           // --------------------------------------------------------
           // STEP 0
           // Калібровка неактивна
           // --------------------------------------------------------
       UINT#0:

           #qx_BlockForward := FALSE;
           #qx_BlockBackward := FALSE;

           IF #StartEdge THEN

               #stat_Calibrated := FALSE;
               #stat_MotionStarted := FALSE;
               #stat_CompletedSteps := DWORD#0;

               // Очищення даних нової процедури калібровки.
               #stat_RawAtReference := DINT#0;
               #stat_RawAtReferenceValid := FALSE;
               #stat_TravelAfterReference_mm := 0.0;

               // Калібровку можна почати тільки після
               // калібровки підйому та в допустимій зоні.
               IF #HoistPositionOK THEN

                   // Нормальний старт перед репером.
                   IF #ix_Reference3K1 THEN
                       #stat_Step := UINT#10;

                       // Якщо механізм знаходиться на / за 3K1,
                       // спочатку необхідно відійти назад.
                   ELSE
                       #stat_Step := UINT#5;
                   END_IF;

               ELSE

                   #stat_Step := UINT#910;

               END_IF;

           END_IF;


           // --------------------------------------------------------
           // STEP 5
           // Попередній відхід назад від 3K1
           // --------------------------------------------------------
       UINT#5:

           #qx_Active := TRUE;

           #qx_BlockForward := TRUE;
           #qx_BlockBackward := FALSE;

           IF #ix_BtnBackward THEN
               #stat_MotionStarted := TRUE;
           END_IF;

           // Після звільнення 3K1 та відпускання кнопки
           // починаємо стандартну процедуру.
           IF #ix_Reference3K1
               AND NOT #ix_BtnBackward
           THEN

               #stat_Step := UINT#10;

           END_IF;


           // --------------------------------------------------------
           // STEP 10
           // Перевірка початкових умов
           // --------------------------------------------------------
       UINT#10:

           #qx_Active := TRUE;

           IF NOT #ix_BtnForward
               AND NOT #ix_BtnBackward
           THEN

               #stat_CompletedSteps.%X0 := TRUE;
               #stat_Step := UINT#20;

           END_IF;


           // --------------------------------------------------------
           // STEP 20
           // Очікування першої команди "Вперед"
           // --------------------------------------------------------
       UINT#20:

           #qx_Active := TRUE;

           #qx_BlockForward := FALSE;
           #qx_BlockBackward := TRUE;

           IF #ix_BtnForward THEN

               #stat_MotionStarted := TRUE;
               #stat_CompletedSteps.%X1 := TRUE;

               #stat_Step := UINT#30;

           END_IF;


           // --------------------------------------------------------
           // STEP 30
           // Перший рух вперед до 3K1
           // --------------------------------------------------------
       UINT#30:

           #qx_Active := TRUE;

           #qx_BlockForward := FALSE;
           #qx_BlockBackward := TRUE;

           IF #ReferenceFalling THEN

               #stat_CompletedSteps.%X2 := TRUE;
               #stat_Step := UINT#40;

           END_IF;


           // --------------------------------------------------------
           // STEP 40
           // Перше проходження 3K1
           // Очікування відпускання кнопки "Вперед"
           // --------------------------------------------------------
       UINT#40:

           #qx_Active := TRUE;

           #qx_BlockForward := TRUE;
           #qx_BlockBackward := TRUE;

           IF NOT #ix_BtnForward THEN

               #stat_CompletedSteps.%X3 := TRUE;
               #stat_Step := UINT#50;

           END_IF;


           // --------------------------------------------------------
           // STEP 50
           // Відхід назад від репера
           // --------------------------------------------------------
       UINT#50:

           #qx_Active := TRUE;

           #qx_BlockForward := TRUE;
           #qx_BlockBackward := FALSE;

           IF #ix_BtnBackward THEN
               #stat_MotionStarted := TRUE;
           END_IF;

           IF #ix_Reference3K1
               AND NOT #ix_BtnBackward
           THEN

               #stat_CompletedSteps.%X4 := TRUE;
               #stat_Step := UINT#60;

           END_IF;


           // --------------------------------------------------------
           // STEP 60
           // Репер звільнений
           // --------------------------------------------------------
       UINT#60:

           #qx_Active := TRUE;

           #qx_BlockForward := TRUE;
           #qx_BlockBackward := TRUE;

           #stat_CompletedSteps.%X5 := TRUE;
           #stat_Step := UINT#70;


           // --------------------------------------------------------
           // STEP 70
           // Очікування повторної команди "Вперед"
           // --------------------------------------------------------
       UINT#70:

           #qx_Active := TRUE;

           #qx_BlockForward := FALSE;
           #qx_BlockBackward := TRUE;

           IF #ix_BtnForward THEN

               #stat_CompletedSteps.%X6 := TRUE;
               #stat_Step := UINT#80;

           END_IF;


           // --------------------------------------------------------
           // STEP 80
           // Повторний точний підхід до 3K1
           // --------------------------------------------------------
       UINT#80:

           #qx_Active := TRUE;

           #qx_BlockForward := FALSE;
           #qx_BlockBackward := TRUE;

           IF #ReferenceFalling THEN

               // У момент спадного фронту 3K1 запам'ятовуємо
               // фактичне raw-положення енкодера.
               IF #ix_PositionScaleValid THEN

                   #stat_RawAtReference :=
                   #id_ActualPositionRaw;

                   #stat_RawAtReferenceValid :=
                   TRUE;

                   #stat_CompletedSteps.%X7 :=
                   TRUE;

                   #stat_Step :=
                   UINT#90;

               ELSE

                   // Масштабування положення невалідне.
                   #stat_RawAtReferenceValid :=
                   FALSE;

                   #stat_Step :=
                   UINT#910;

               END_IF;

           END_IF;



           // --------------------------------------------------------
           // STEP 90
           // Quick Stop
           // --------------------------------------------------------
       UINT#90:

           #qx_Active := TRUE;

           #qx_BlockForward := TRUE;
           #qx_BlockBackward := TRUE;
           #qx_QuickStop := TRUE;

           #stat_CompletedSteps.%X8 := TRUE;

           #stat_Step := UINT#100;


           // --------------------------------------------------------
           // STEP 100
           // Очікування повної зупинки ПЧ
           // --------------------------------------------------------
       UINT#100:

           #qx_Active := TRUE;

           #qx_BlockForward := TRUE;
           #qx_BlockBackward := TRUE;

           // Quick Stop утримується до підтвердженої зупинки.
           #qx_QuickStop := TRUE;

           IF #qx_DriveStandstill
               AND NOT #ix_BtnForward
               AND NOT #ix_BtnBackward
           THEN

               // Для розрахунку повинна бути зафіксована
               // точка 3K1 і валідне масштабування.
               IF #stat_RawAtReferenceValid
                   AND #ix_PositionScaleValid
               THEN

                   // Розрахунок шляху, пройденого від моменту
                   // спрацювання 3K1 до повної зупинки.
                   #stat_TravelAfterReference_mm :=
                   (
                   DINT_TO_LREAL(#id_ActualPositionRaw)
                   - DINT_TO_LREAL(#stat_RawAtReference)
                   )
                   * #il_Scale_mm_per_count;

                   #stat_CompletedSteps.%X9 :=
                   TRUE;

                   #stat_Step :=
                   UINT#110;

               ELSE

                   // Немає валідної реперної точки
                   // або масштабування положення.
                   #stat_Step :=
                   UINT#910;

               END_IF;

           END_IF;



           // --------------------------------------------------------
           // STEP 110
           // Запуск preset
           // --------------------------------------------------------
       UINT#110:

           #qx_Active := TRUE;

           #qx_BlockForward := TRUE;
           #qx_BlockBackward := TRUE;

           #qx_PresetServiceEnable := TRUE;

           #qx_PresetPermit :=
           #qx_DriveStandstill
           AND NOT #ix_BtnForward
           AND NOT #ix_BtnBackward
           AND #ix_EncoderReady
           AND NOT #ix_EncoderFault
           AND NOT #ix_DriveFault;

           IF #qx_PresetPermit THEN

               #qx_PresetStart := TRUE;

               #stat_CompletedSteps.%X10 := TRUE;
               #stat_Step := UINT#120;

           END_IF;


           // --------------------------------------------------------
           // STEP 120
           // Очікування завершення preset
           // --------------------------------------------------------
       UINT#120:

           #qx_Active := TRUE;

           #qx_BlockForward := TRUE;
           #qx_BlockBackward := TRUE;

           #qx_PresetServiceEnable := TRUE;

           #qx_PresetPermit :=
           #qx_DriveStandstill
           AND NOT #ix_BtnForward
           AND NOT #ix_BtnBackward
           AND NOT #ix_EncoderFault
           AND NOT #ix_DriveFault;

           IF #ix_PresetDone THEN

               #stat_CompletedSteps.%X11 := TRUE;
               #stat_Step := UINT#130;

           ELSIF #ix_PresetError THEN

               #stat_Step := UINT#910;

           END_IF;


           // --------------------------------------------------------
           // STEP 130
           // Калібровка успішно завершена
           // --------------------------------------------------------
       UINT#130:

           #qx_BlockForward := FALSE;
           #qx_BlockBackward := FALSE;

           #stat_Calibrated := TRUE;
           #stat_CompletedSteps.%X12 := TRUE;


           // --------------------------------------------------------
           // STEP 900
           // Ручне переривання
           // --------------------------------------------------------
       UINT#900:

           #qx_Aborted := TRUE;

           #qx_BlockForward := TRUE;
           #qx_BlockBackward := TRUE;

           #qx_QuickStop := TRUE;


           // --------------------------------------------------------
           // STEP 910
           // Помилка процедури
           // --------------------------------------------------------
       UINT#910:

           #qx_Fault := TRUE;

           #qx_BlockForward := TRUE;
           #qx_BlockBackward := TRUE;

           #qx_QuickStop := TRUE;


       ELSE

           #stat_Step := UINT#910;

   END_CASE;


   // ============================================================
   // 11. Основні статуси
   // ============================================================

   #qu_CurrentStep :=
   #stat_Step;

   #qd_CompletedSteps :=
   #stat_CompletedSteps;

   #qx_Calibrated :=
   #stat_Calibrated
   OR #ix_ForceCalibrated;

   // Шлях від повторного проходження 3K1
   // до підтвердженої повної зупинки.
   #ql_TravelAfterReference_mm :=
   #stat_TravelAfterReference_mm;

   // ============================================================
   // 12. Активний таймер для HMI
   // ============================================================

   #qt_ActiveTimerElapsed := T#0ms;
   #qt_ActiveTimerPreset := T#0ms;
   #qt_ActiveTimerRemaining := T#0ms;

   // Timeout A
   IF (#stat_Step = UINT#5)
       OR (#stat_Step = UINT#20)
       OR (#stat_Step = UINT#50)
       OR (#stat_Step = UINT#70)
   THEN

       #qt_ActiveTimerElapsed :=
       #tmr_TimeoutA.ET;

       #qt_ActiveTimerPreset :=
       #it_TimeoutA;

       IF #tmr_TimeoutA.ET < #it_TimeoutA THEN

           #qt_ActiveTimerRemaining :=
           #it_TimeoutA - #tmr_TimeoutA.ET;

       END_IF;


       // Timeout B
   ELSIF 
       (#stat_Step = UINT#30)
       OR (#stat_Step = UINT#80)
   THEN

       #qt_ActiveTimerElapsed :=
       #tmr_TimeoutB.ET;

       #qt_ActiveTimerPreset :=
       #it_TimeoutB;

       IF #tmr_TimeoutB.ET < #it_TimeoutB THEN

           #qt_ActiveTimerRemaining :=
           #it_TimeoutB - #tmr_TimeoutB.ET;

       END_IF;


       // Standstill
   ELSIF #stat_Step = UINT#100 THEN

       #qt_ActiveTimerElapsed :=
       #tmr_Standstill.ET;

       #qt_ActiveTimerPreset :=
       #it_StandstillConfirm;

       IF #tmr_Standstill.ET < #it_StandstillConfirm THEN

           #qt_ActiveTimerRemaining :=
           #it_StandstillConfirm - #tmr_Standstill.ET;

       END_IF;

   END_IF;


   // ============================================================
   // 13. Діагностичне слово
   // ============================================================

   #qw_Status := W#16#0000;

   IF #qx_Active THEN
       #qw_Status := #qw_Status OR W#16#0001;
   END_IF;

   IF #qx_Calibrated THEN
       #qw_Status := #qw_Status OR W#16#0002;
   END_IF;

   IF #qx_Aborted THEN
       #qw_Status := #qw_Status OR W#16#0004;
   END_IF;

   IF #qx_Fault THEN
       #qw_Status := #qw_Status OR W#16#0008;
   END_IF;

   IF #qx_DriveStandstill THEN
       #qw_Status := #qw_Status OR W#16#0010;
   END_IF;

   IF #ix_PresetBusy THEN
       #qw_Status := #qw_Status OR W#16#0020;
   END_IF;

   IF #ix_PresetError THEN
       #qw_Status := #qw_Status OR W#16#0040;
   END_IF;

   IF #tmr_TimeoutA.Q THEN
       #qw_Status := #qw_Status OR W#16#0100;
   END_IF;

   IF #tmr_TimeoutB.Q THEN
       #qw_Status := #qw_Status OR W#16#0200;
   END_IF;

   IF #ix_DriveFault THEN
       #qw_Status := #qw_Status OR W#16#0400;
   END_IF;

   IF #ix_EncoderFault THEN
       #qw_Status := #qw_Status OR W#16#0800;
   END_IF;

   IF NOT #ix_EncoderReady THEN
       #qw_Status := #qw_Status OR W#16#1000;
   END_IF;


   // ============================================================
   // 14. Запам'ятовування станів
   // ============================================================

   #stat_StartOld :=
   #ix_Start;

   #stat_ResetOld :=
   #ix_Reset;

   #stat_AbortOld :=
   #ix_Abort;

   #stat_ReferenceOld :=
   #ix_Reference3K1;
END_FUNCTION_BLOCK

FUNCTION_BLOCK "FB_TrolleyCalibrationDiag"   // FB712, SCL
{ S7_Optimized_Access := 'TRUE' }
VERSION : 0.1
   VAR_INPUT
      ix_Reset : Bool := FALSE;   // Скидання зафіксованих діагностичних помилок
      ix_EncoderReady : Bool := FALSE;   // Енкодер 3BR готовий
      ix_EncoderFault : Bool := FALSE;   // Помилка енкодера
      ix_CommunicationFault : Bool := FALSE;   // Помилка зв'язку з енкодером
      il_Position_mm : LReal := 0.0;   // Поточна координата візка, мм
      ix_MoveCommand : Bool := FALSE;   // Дійсна команда руху візка
      ix_DriveFault : Bool := FALSE;   // Аварія привода
      ir_DriveVelocity_rpm : Real := 0.0;   // Фактична швидкість привода
      ix_CalibrationActive : Bool := FALSE;   // Процедура калібровки візка активна
      ix_Calibrated : Bool := FALSE;   // Візок відкалібрований
      ix_ManualDriveActive : Bool := FALSE;   // Ручний привод активний; поки FALSE
      il_NoMoveThreshold_mm : LReal := 5.0;   // Допустима зміна положення без команди
      il_MoveMinDelta_mm : LReal := 1.0;   // Мінімальна зміна при русі
      it_MoveUpdateTimeout : Time := T#1s;   // Максимальний час без зміни положення
      ir_StandstillSpeed_rpm : Real := 5.0;   // Поріг повної зупинки
      it_StandstillConfirm : Time := T#500ms;   // Час підтвердження повної зупинки
      il_StartupTolerance_mm : LReal := 5.0;   // Допуск після запуску PLC
   END_VAR
   VAR_OUTPUT
      qx_EncoderControlHealthy : Bool := FALSE;   // Енкодер 3BR і зв'язок справні
      qx_StartupDataConsistent : Bool := TRUE;   // Положення після старту PLC узгоджене
      qx_NoMovementWithoutCommand : Bool := TRUE;   // Не виявлено переміщення без команди
      qx_NoManualMovementDetected : Bool := TRUE;   // Не виявлено нештатного руху без ручного приводу
      qx_EncoderUpdatesDuringMotion : Bool := TRUE;   // Енкодер змінює значення при команді руху
      qx_EncoderReplacementNotDetected : Bool := TRUE;   // Зарезервовано; поки завжди норма
      qx_DiagnosticsHealthy : Bool := FALSE;   // Усі реалізовані контролі в нормі
      qx_DriveStandstill : Bool := FALSE;   // Підтверджена повна зупинка
      ql_PositionDeltaStopped_mm : LReal := 0.0;   // Зміна позиції від точки зупинки
      ql_PositionDeltaMotion_mm : LReal := 0.0;   // Зміна позиції для watchdog руху
   END_VAR
   VAR RETAIN
      stat_SavedPosition_mm : LReal := 0.0;   // Положення, збережене до перезапуску
      stat_SavedPositionValid : Bool := FALSE;   // Ознака валідності збереженого положення
   END_VAR
   VAR
      stat_StartupChecked : Bool := FALSE;   // Перевірка після запуску PLC виконана
      stat_StopReference_mm : LReal := 0.0;   // Базова позиція після зупинки
      stat_StopReferenceValid : Bool := FALSE;   // Базова позиція зупинки валідна
      stat_MoveReference_mm : LReal := 0.0;   // Базова позиція для watchdog руху
      stat_MoveMonitorActive : Bool := FALSE;   // Контроль зміни позиції при русі активний
      stat_WasMoving : Bool := FALSE;   // Ознака, що механізм до цього рухався
      stat_StartupMismatchFault : Bool := FALSE;   // Виявлена невідповідність положення після запуску
      stat_MoveWithoutCommandFault : Bool := FALSE;   // Виявлено зміну положення без команди руху
      stat_NoUpdateDuringMotionFault : Bool := FALSE;   // Не виявлено зміни положення при команді руху
      stat_CalibratedOld : Bool := FALSE;   // Попередній стан сигналу Calibrated
      tmr_Standstill : TON_TIME;   // Таймер підтвердження повної зупинки
      tmr_MoveUpdate : TON_TIME;   // Watchdog оновлення положення при русі
   END_VAR
   VAR_TEMP
      EncoderHealthy : Bool;   // Поточна справність енкодера і зв'язку
      StandstillCondition : Bool;   // Умова низької швидкості
      CalibratedRising : Bool;   // Передній фронт статусу калібровки
      MoveDeltaReached : Bool;   // Досягнута мінімальна зміна положення
      MoveWatchdogEnable : Bool;   // Дозвіл watchdog руху
   END_VAR
BEGIN
       // ============================================================
       // 1. Загальна справність енкодера 3BR
       // ============================================================

       #EncoderHealthy :=
       #ix_EncoderReady
       AND NOT #ix_EncoderFault
       AND NOT #ix_CommunicationFault;

       #qx_EncoderControlHealthy :=
       #EncoderHealthy;


       // ============================================================
       // 2. Визначення повної зупинки
       // ============================================================

       #StandstillCondition :=
       ABS(#ir_DriveVelocity_rpm)
       <= #ir_StandstillSpeed_rpm;

       #tmr_Standstill(
                       IN :=
                       #StandstillCondition
                       AND NOT #ix_MoveCommand,
                       PT := #it_StandstillConfirm
       );

       #qx_DriveStandstill :=
       #tmr_Standstill.Q;


       // ============================================================
       // 3. Фронт отримання статусу "Калібровано"
       // ============================================================

       #CalibratedRising :=
       #ix_Calibrated
       AND NOT #stat_CalibratedOld;


       // ============================================================
       // 4. Reset діагностики
       // ============================================================

       IF #ix_Reset THEN

           #stat_StartupMismatchFault := FALSE;
           #stat_MoveWithoutCommandFault := FALSE;
           #stat_NoUpdateDuringMotionFault := FALSE;

           #stat_StopReferenceValid := FALSE;
           #stat_MoveMonitorActive := FALSE;

       END_IF;


       // ============================================================
       // 5. Перевірка положення після запуску PLC
       //
       // Виконується один раз після появи валідних даних енкодера.
       // Retain-позиція не перезаписується до завершення перевірки.
       // ============================================================

       IF NOT #stat_StartupChecked
           AND #EncoderHealthy
       THEN

           IF #stat_SavedPositionValid THEN

               IF ABS(#il_Position_mm - #stat_SavedPosition_mm)
                   > #il_StartupTolerance_mm
               THEN

                   #stat_StartupMismatchFault := TRUE;

               END_IF;

           ELSE

               // Перший запуск: попереднього значення ще немає.
               #stat_SavedPosition_mm :=
               #il_Position_mm;

               #stat_SavedPositionValid := TRUE;

           END_IF;

           #stat_StartupChecked := TRUE;

           // Початкова база для контролю нерухомості.
           #stat_StopReference_mm :=
           #il_Position_mm;

           #stat_StopReferenceValid := TRUE;

       END_IF;


       // ============================================================
       // 6. Після успішної калібровки
       //
       // Preset штатно змінює координату без фізичного руху.
       // Тому після калібровки формуємо нову базову позицію.
       // ============================================================

       IF #CalibratedRising
           AND #EncoderHealthy
       THEN

           #stat_StopReference_mm :=
           #il_Position_mm;

           #stat_StopReferenceValid := TRUE;

           #stat_SavedPosition_mm :=
           #il_Position_mm;

           #stat_SavedPositionValid := TRUE;

           // Калібровка формує нову достовірну координату.
           #stat_StartupMismatchFault := FALSE;
           #stat_MoveWithoutCommandFault := FALSE;
           #stat_NoUpdateDuringMotionFault := FALSE;

       END_IF;


       // ============================================================
       // 7. Запам'ятовування факту руху
       // ============================================================

       IF #ix_MoveCommand THEN
           #stat_WasMoving := TRUE;
       END_IF;


       // ============================================================
       // 8. Формування нової бази після завершення руху
       //
       // Після підтвердженої повної зупинки зберігаємо положення.
       // ============================================================

       IF #qx_DriveStandstill
           AND #stat_WasMoving
           AND #EncoderHealthy
           AND NOT #ix_CalibrationActive
       THEN

           #stat_StopReference_mm :=
           #il_Position_mm;

           #stat_StopReferenceValid := TRUE;

           #stat_SavedPosition_mm :=
           #il_Position_mm;

           #stat_SavedPositionValid := TRUE;

           #stat_WasMoving := FALSE;

       END_IF;


       // ============================================================
       // 9. Контроль зміни положення без команди руху
       //
       // Контроль виконується тільки:
       // - після підтвердженої повної зупинки;
       // - без команди руху;
       // - без ручного приводу;
       // - поза процедурою калібровки.
       // ============================================================

       #ql_PositionDeltaStopped_mm := 0.0;

       IF #qx_DriveStandstill
           AND NOT #ix_MoveCommand
           AND NOT #ix_ManualDriveActive
           AND NOT #ix_CalibrationActive
           AND #EncoderHealthy
           AND #stat_StopReferenceValid
       THEN

           #ql_PositionDeltaStopped_mm :=
           ABS(#il_Position_mm - #stat_StopReference_mm);

           IF #ql_PositionDeltaStopped_mm
               > #il_NoMoveThreshold_mm
           THEN

               #stat_MoveWithoutCommandFault := TRUE;

           END_IF;

       END_IF;


       // ============================================================
       // 10. Контроль оновлення енкодера під час руху
       //
       // Якщо є дійсна команда руху і немає аварії привода,
       // координата повинна змінюватись не менш ніж на задану
       // величину протягом MoveUpdateTimeout.
       // ============================================================

       IF #ix_MoveCommand
           AND NOT #ix_DriveFault
           AND #EncoderHealthy
       THEN

           IF NOT #stat_MoveMonitorActive THEN

               #stat_MoveReference_mm :=
               #il_Position_mm;

               #stat_MoveMonitorActive := TRUE;

           END_IF;

           #ql_PositionDeltaMotion_mm :=
           ABS(#il_Position_mm - #stat_MoveReference_mm);

           #MoveDeltaReached :=
           #ql_PositionDeltaMotion_mm >= #il_MoveMinDelta_mm;

           IF #MoveDeltaReached THEN

               // Є нормальна зміна координати.
               // Починаємо наступний інтервал контролю.
               #stat_MoveReference_mm :=
               #il_Position_mm;

           END_IF;

       ELSE

           #stat_MoveMonitorActive := FALSE;
           #ql_PositionDeltaMotion_mm := 0.0;
           #MoveDeltaReached := FALSE;

       END_IF;


       // Watchdog працює, поки координата не змінилася
       // на необхідну величину.
       #MoveWatchdogEnable :=
       #stat_MoveMonitorActive
       AND NOT #MoveDeltaReached;

       #tmr_MoveUpdate(
                       IN := #MoveWatchdogEnable,
                       PT := #it_MoveUpdateTimeout
       );

       IF #tmr_MoveUpdate.Q THEN
           #stat_NoUpdateDuringMotionFault := TRUE;
       END_IF;


       // ============================================================
       // 11. Позитивні діагностичні виходи
       // ============================================================

       #qx_StartupDataConsistent :=
       NOT #stat_StartupMismatchFault;

       #qx_NoMovementWithoutCommand :=
       NOT #stat_MoveWithoutCommandFault;

       // Поки окремого сигналу ручного приводу немає.
       // Контроль використовує його як дозвільну умову.
       #qx_NoManualMovementDetected :=
       NOT #stat_MoveWithoutCommandFault;

       #qx_EncoderUpdatesDuringMotion :=
       NOT #stat_NoUpdateDuringMotionFault;


       // ============================================================
       // 12. Контроль фізичної заміни енкодера
       //
       // Поки не реалізований.
       // До появи надійного способу ідентифікації енкодера
       // сигнал примусово встановлений у стан "Норма".
       // ============================================================

       #qx_EncoderReplacementNotDetected := TRUE;


       // ============================================================
       // 13. Загальний результат
       // ============================================================

       #qx_DiagnosticsHealthy :=
       #qx_EncoderControlHealthy
       AND #qx_StartupDataConsistent
       AND #qx_NoMovementWithoutCommand
       AND #qx_NoManualMovementDetected
       AND #qx_EncoderUpdatesDuringMotion;


       // ============================================================
       // 14. Запам'ятовування станів
       // ============================================================

       #stat_CalibratedOld :=
       #ix_Calibrated;
END_FUNCTION_BLOCK

// folder: 70_FireAlarm

FUNCTION_BLOCK "FB_FireAlarm"   // FB70, LAD
TITLE = Пожежна сигналізація
{ S7_Optimized_Access := 'TRUE' }
VERSION : 0.1
   VAR_INPUT
      ix_VFD1_PM_AirIntakeOvertemp : Bool;   // ПЧ1 - Силовий модуль: перегрів повітря на вході
      ix_VFD2_PM_AirIntakeOvertemp : Bool;   // ПЧ2 - Силовий модуль: перегрів повітря на вході
      ix_VFD3_PM_AirIntakeOvertemp : Bool;   // ПЧ3 - Силовий модуль: перегрів повітря на вході
      ix_VFD1_OvertempMonitor : Bool;   // ПЧ1 - Додатковий контроль температури
      ix_VFD2_OvertempMonitor : Bool;   // ПЧ2 - Додатковий контроль температури
      ix_VFD3_OvertempMonitor : Bool;   // ПЧ3 - Додатковий контроль температури
      ix_Ack : Bool;   // Скидання пожежної сигналізації
   END_VAR
   VAR_OUTPUT
      ox_FireAlarmActive : Bool;   // Активна пожежна сигналізація
      ox_SoundFireAlarm : Bool;   // Звукова пожежна сигналізація
   END_VAR
   VAR
      T_FireAlarmDelay : TON_TIME;   // Таймер затримки спрацювання сигналізації
      T_DelaySP : Time := T#30s;   // Уставка часу
      T_SoundAlarm_Active : TON_TIME;   // Таймер видачі звуку
      T_SoundAlarm_Idle : TON_TIME;   // Таймер паузи звуку
      sx_SoundAlarmActive : Bool;   // Активна звукова сигналызація
   END_VAR
   VAR_TEMP
      Condition1 : Bool;   // Умова 1 = ПЧ1+ПЧ2
      Condition2 : Bool;   // Умова 2 = ПЧ1 +ПЧ3
      Condition3 : Bool;   // Умова 3 = ПЧ2 + ПЧ3
   END_VAR
   // T_SoundAlarm_Active.PT := T#3s;
   // T_SoundAlarm_Idle.PT := T#1s;
BEGIN

REGION Network 1: Скидання активної пожежної сигналізації
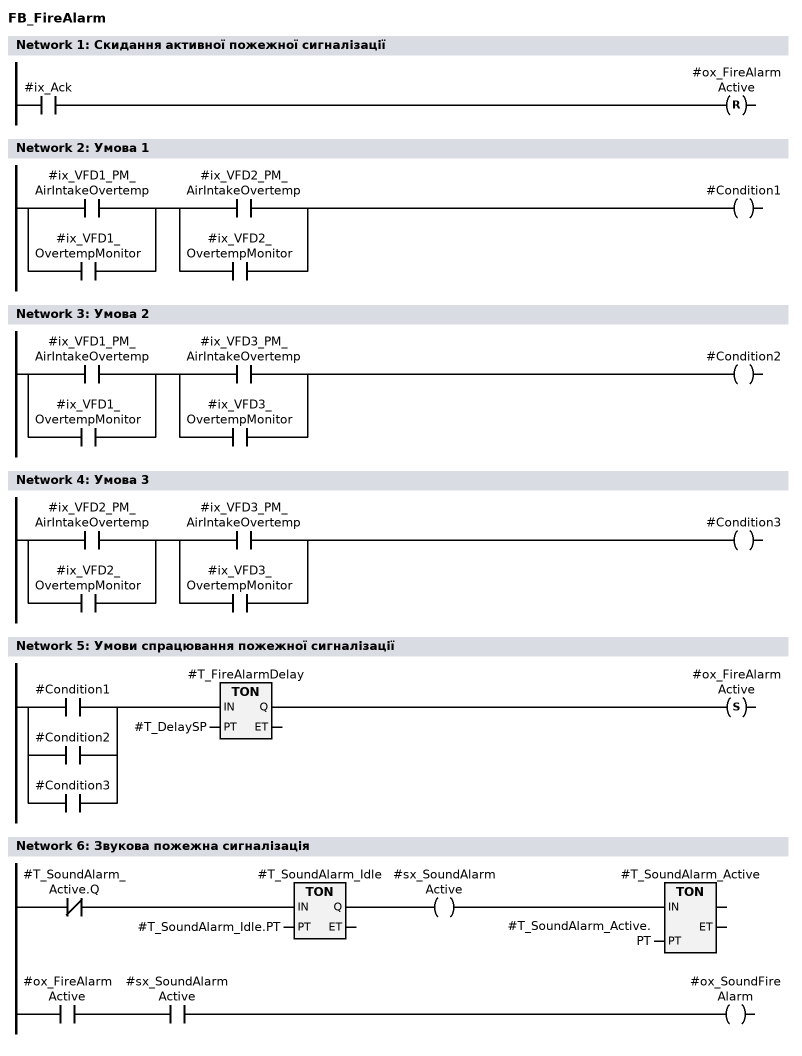
   RUNG wire#powerrail
      Contact( #ix_Ack )
      R_Coil( #ox_FireAlarmActive )
   END_RUNG
   // the same network as SCL:
   IF #ix_Ack THEN #ox_FireAlarmActive := FALSE; END_IF;
END_REGION

REGION Network 2: Умова 1
   RUNG wire#powerrail
      Contact( #ix_VFD1_PM_AirIntakeOvertemp )
      wire#w1
      Contact( #ix_VFD2_PM_AirIntakeOvertemp )
      wire#w2
      Coil( #Condition1 )
   END_RUNG
   RUNG wire#powerrail
      Contact( #ix_VFD1_OvertempMonitor )
   END_RUNG wire#w1
   RUNG wire#w1
      Contact( #ix_VFD2_OvertempMonitor )
   END_RUNG wire#w2
   // the same network as SCL:
   #Condition1 := (#ix_VFD1_PM_AirIntakeOvertemp OR #ix_VFD1_OvertempMonitor) AND (#ix_VFD2_PM_AirIntakeOvertemp OR #ix_VFD2_OvertempMonitor);
END_REGION

REGION Network 3: Умова 2
   RUNG wire#powerrail
      Contact( #ix_VFD1_PM_AirIntakeOvertemp )
      wire#w1
      Contact( #ix_VFD3_PM_AirIntakeOvertemp )
      wire#w2
      Coil( #Condition2 )
   END_RUNG
   RUNG wire#powerrail
      Contact( #ix_VFD1_OvertempMonitor )
   END_RUNG wire#w1
   RUNG wire#w1
      Contact( #ix_VFD3_OvertempMonitor )
   END_RUNG wire#w2
   // the same network as SCL:
   #Condition2 := (#ix_VFD1_PM_AirIntakeOvertemp OR #ix_VFD1_OvertempMonitor) AND (#ix_VFD3_PM_AirIntakeOvertemp OR #ix_VFD3_OvertempMonitor);
END_REGION

REGION Network 4: Умова 3
   RUNG wire#powerrail
      Contact( #ix_VFD2_PM_AirIntakeOvertemp )
      wire#w1
      Contact( #ix_VFD3_PM_AirIntakeOvertemp )
      wire#w2
      Coil( #Condition3 )
   END_RUNG
   RUNG wire#powerrail
      Contact( #ix_VFD2_OvertempMonitor )
   END_RUNG wire#w1
   RUNG wire#w1
      Contact( #ix_VFD3_OvertempMonitor )
   END_RUNG wire#w2
   // the same network as SCL:
   #Condition3 := (#ix_VFD2_PM_AirIntakeOvertemp OR #ix_VFD2_OvertempMonitor) AND (#ix_VFD3_PM_AirIntakeOvertemp OR #ix_VFD3_OvertempMonitor);
END_REGION

REGION Network 5: Умови спрацювання пожежної сигналізації
   #T_FireAlarmDelay(IN := #Condition1 OR #Condition2 OR #Condition3, PT := #T_DelaySP);   // TON
   IF #T_FireAlarmDelay.Q THEN #ox_FireAlarmActive := TRUE; END_IF;
END_REGION

REGION Network 6: Звукова пожежна сигналізація
   #T_SoundAlarm_Idle(IN := NOT #T_SoundAlarm_Active.Q, PT := #T_SoundAlarm_Idle.PT);   // TON
   #sx_SoundAlarmActive := #T_SoundAlarm_Idle.Q;
   #T_SoundAlarm_Active(IN := #T_SoundAlarm_Idle.Q, PT := #T_SoundAlarm_Active.PT);   // TON
   #ox_SoundFireAlarm := #ox_FireAlarmActive AND #sx_SoundAlarmActive;
END_REGION
END_FUNCTION_BLOCK

FUNCTION "FC_FireAlarmCall" : Void   // FC70, LAD
TITLE = Пожежна сигналізація
{ S7_Optimized_Access := 'TRUE' }
VERSION : 0.1
BEGIN

REGION Network 1: Пожежна сигналізація
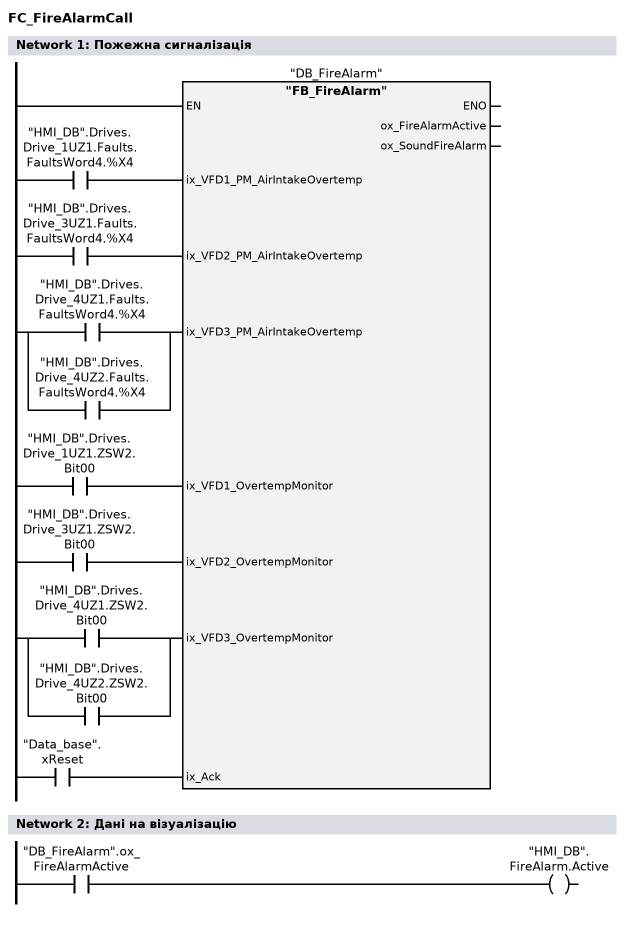
   RUNG wire#powerrail
      "DB_FireAlarm"(ix_VFD1_PM_AirIntakeOvertemp := wire#w1, ix_VFD2_PM_AirIntakeOvertemp := wire#w2, ix_VFD3_PM_AirIntakeOvertemp := wire#w3, ix_VFD1_OvertempMonitor := wire#w4, ix_VFD2_OvertempMonitor := wire#w5, ix_VFD3_OvertempMonitor := wire#w6, ix_Ack := wire#w7, ox_FireAlarmActive =>, ox_SoundFireAlarm =>)
   END_RUNG
   RUNG wire#powerrail
      Contact( "HMI_DB".Drives.Drive_1UZ1.Faults.FaultsWord4.%X4 )
   END_RUNG wire#w1
   RUNG wire#powerrail
      Contact( "HMI_DB".Drives.Drive_3UZ1.Faults.FaultsWord4.%X4 )
   END_RUNG wire#w2
   RUNG wire#powerrail
      Contact( "HMI_DB".Drives.Drive_4UZ1.Faults.FaultsWord4.%X4 )
   END_RUNG wire#w3
   RUNG wire#powerrail
      Contact( "HMI_DB".Drives.Drive_4UZ2.Faults.FaultsWord4.%X4 )
   END_RUNG wire#w3
   RUNG wire#powerrail
      Contact( "HMI_DB".Drives.Drive_1UZ1.ZSW2.Bit00 )
   END_RUNG wire#w4
   RUNG wire#powerrail
      Contact( "HMI_DB".Drives.Drive_3UZ1.ZSW2.Bit00 )
   END_RUNG wire#w5
   RUNG wire#powerrail
      Contact( "HMI_DB".Drives.Drive_4UZ1.ZSW2.Bit00 )
   END_RUNG wire#w6
   RUNG wire#powerrail
      Contact( "HMI_DB".Drives.Drive_4UZ2.ZSW2.Bit00 )
   END_RUNG wire#w6
   RUNG wire#powerrail
      Contact( "Data_base".xReset )
   END_RUNG wire#w7
   // the same network as SCL:
   "DB_FireAlarm"(ix_VFD1_PM_AirIntakeOvertemp := "HMI_DB".Drives.Drive_1UZ1.Faults.FaultsWord4.%X4,   // "FB_FireAlarm"
                  ix_VFD2_PM_AirIntakeOvertemp := "HMI_DB".Drives.Drive_3UZ1.Faults.FaultsWord4.%X4,
                  ix_VFD3_PM_AirIntakeOvertemp := "HMI_DB".Drives.Drive_4UZ1.Faults.FaultsWord4.%X4 OR "HMI_DB".Drives.Drive_4UZ2.Faults.FaultsWord4.%X4,
                  ix_VFD1_OvertempMonitor := "HMI_DB".Drives.Drive_1UZ1.ZSW2.Bit00,
                  ix_VFD2_OvertempMonitor := "HMI_DB".Drives.Drive_3UZ1.ZSW2.Bit00,
                  ix_VFD3_OvertempMonitor := "HMI_DB".Drives.Drive_4UZ1.ZSW2.Bit00 OR "HMI_DB".Drives.Drive_4UZ2.ZSW2.Bit00,
                  ix_Ack := "Data_base".xReset);
END_REGION

REGION Network 2: Дані на візуалізацію
   RUNG wire#powerrail
      Contact( "DB_FireAlarm".ox_FireAlarmActive )
      Coil( "HMI_DB".FireAlarm.Active )
   END_RUNG
   // the same network as SCL:
   "HMI_DB".FireAlarm.Active := "DB_FireAlarm".ox_FireAlarmActive;
END_REGION
END_FUNCTION

// folder: 80_Encoders

FUNCTION_BLOCK "FB_Enc_Tlg89_Com"   // FB80, SCL
{ S7_Optimized_Access := 'TRUE' }
VERSION : 0.1
   VAR_INPUT
      HW_ID_Tlg89 : Hw_Io;   // HW ID підмодуля Standard Telegram 89, PZD3/5. Це має бути HW ID саме телеграмного підмодуля, не головного модуля енкодера.
      Enable : Bool := TRUE;   // Загальний дозвіл роботи блока.
      AckError : Bool := FALSE;   // Квітування помилки енкодера по передньому фронту. Формує STW2_ENC bit 7.
      PresetServiceEnable : Bool := FALSE;   // Дозвіл сервісної функції preset. Для нормальної роботи має бути FALSE.
      PresetPermit : Bool := FALSE;   // Додатковий дозвіл preset від логіки ПЛК. Сюди треба подавати умови: механізм стоїть, сервісний режим активний, немає команд руху.
      PresetStart : Bool := FALSE;   // Команда запуску preset по передньому фронту. Формує STW2_ENC bit 0.
      PresetValueRaw : DInt := DINT#0;   // Значення preset у raw-count. Для 30-bit енкодера допустимий діапазон 0...1073741823.
      SimulationMode : Bool := FALSE;   // Дозвіл режиму симуляції з боку виклику блока.
      SimPzdIn : "UDT_Enc_Tlg89_In";   // Вхідна PZD-структура від симулятора енкодера.
      SimInputValid : Bool := FALSE;   // Ознака, що симуляційні PZD-дані достовірні.
   END_VAR
   VAR_OUTPUT
      AbsolutePositionRaw : DInt := DINT#0;   // Абсолютне положення з G1_XIST2. Використовувати тільки якщо PositionDataValid = TRUE.
      VelocityRaw : DInt := DINT#0;   // Швидкість з NIST_B. Використовувати тільки якщо VelocityDataValid = TRUE.
      PositionDataValid : Bool := FALSE;   // Положення можна використовувати в логіці керування.
      VelocityDataValid : Bool := FALSE;   // Швидкість можна використовувати в логіці керування.
      EncoderReady : Bool := FALSE;   // Фінальна готовність енкодера для логіки крана.
      CommunicationFault : Bool := FALSE;   // Загальна помилка комунікації або недостовірності обміну.
      EncoderFault : Bool := FALSE;   // ZSW2_ENC bit 3. Активна помилка енкодера.
      EncoderAlarm : Bool := FALSE;   // ZSW2_ENC bit 7. Попередження або alarm.
      EncoderErrorCode : DInt := DINT#0;   // Код активної помилки енкодера з G1_XIST2. 0 — активної помилки немає.
      ControlByPlcActive : Bool := FALSE;   // ZSW2_ENC bit 9. Енкодер підтвердив керування / валідність циклічних даних від PLC.
      EncoderLifeValid : Bool := FALSE;   // Encoder sign-of-life валідний.
      PresetBusy : Bool := FALSE;   // TRUE, якщо preset-процедура активна.
      PresetDone : Bool := FALSE;   // Імпульс на один цикл після успішного preset.
      PresetError : Bool := FALSE;   // TRUE, якщо preset-процедура завершилась помилкою.
      PresetStatus : Word := W#16#0000;   // Діагностичний код preset-процедури.
      Status : Word := W#16#0000;   // Загальне діагностичне слово блока.
   END_VAR
   VAR
      SimulationPermit : Bool := FALSE;   // Додатковий дозвіл симуляції. Реальна симуляція активна тільки якщо SimulationMode = TRUE і SimulationPermit = TRUE.
      EnableSignOfLife : Bool := FALSE;   // Дозвіл формування master sign-of-life у STW2_ENC bits 12...15.
      MonitorSignOfLife : Bool := FALSE;   // Дозвіл контролю encoder sign-of-life із ZSW2_ENC bits 12...15.
      MaxUnchangedLifeCycles : UInt := UINT#10;   // Максимальна кількість циклів без зміни encoder sign-of-life.
   END_VAR
   VAR RETAIN
      MaxPositionRaw : DInt := DINT#1073741823;   // Максимальне допустиме raw-значення для 30-bit енкодера.
   END_VAR
   VAR
      PzdIn : "UDT_Enc_Tlg89_In";   // Буфер для DPRD_DAT у реальному режимі.
      PzdOut : "UDT_Enc_Tlg89_Out";   // Буфер для DPWR_DAT у реальному режимі.
      PzdInActual : "UDT_Enc_Tlg89_In";   // Фактично використана вхідна PZD-структура: з енкодера або з симулятора.
      PzdOutActual : "UDT_Enc_Tlg89_Out";   // Фактично сформована вихідна PZD-структура.
      SimPzdOut : "UDT_Enc_Tlg89_Out";   // Вихідна PZD-структура для симулятора. Підключається до входу PzdFromController у симуляційному FB.
      ReadRetVal : Int := INT#0;   // Код повернення DPRD_DAT.
      WriteRetVal : Int := INT#0;   // Код повернення DPWR_DAT.
      ReadError : Bool := FALSE;   // Помилка читання PZD-даних.
      WriteError : Bool := FALSE;   // Помилка запису PZD-даних.
      PresetAck : Bool := FALSE;   // ZSW2_ENC bit 0. Підтвердження виконання preset.
      PositionActualValidBit : Bool := FALSE;   // ZSW2_ENC bit 1. Фактичне положення валідне.
      VelocityActualValidBit : Bool := FALSE;   // ZSW2_ENC bit 2. Фактична швидкість валідна.
      MasterSignOfLife : USInt := USINT#1;   // Поточне значення master sign-of-life, яке PLC передає в STW2_ENC bits 12...15.
      EncoderSignOfLife : USInt := USINT#0;   // Поточне значення encoder sign-of-life із ZSW2_ENC bits 12...15.
      EncoderLifeChanged : Bool := FALSE;   // Encoder sign-of-life змінився в поточному циклі.
      UnchangedLifeCycles : UInt := UINT#0;   // Кількість циклів без зміни encoder sign-of-life.
   END_VAR
   VAR RETAIN
      ActivePresetValueRaw : DInt := DINT#0;   // Значення, яке зараз передається в G1_XIST_PRESET_B1.
   END_VAR
   VAR
      PrevPresetAck : Bool := FALSE;   // Попередній стан ZSW2_ENC bit 0.
      PresetAckRising : Bool := FALSE;   // Передній фронт підтвердження preset від енкодера.
      AckErrorEdge : R_TRIG;   // Формування переднього фронту AckError.
      PresetStartEdge : R_TRIG;   // Формування переднього фронту PresetStart.
      SimulationActive : Bool := FALSE;   // Активний режим симуляції: SimulationMode AND SimulationPermit.
      MasterLifeCounter : USInt := USINT#1;   // Внутрішній лічильник master sign-of-life 1...15.
      LastEncoderLifeCounter : USInt := USINT#0;   // Попереднє значення encoder sign-of-life.
      UnchangedLifeCyclesInt : UInt := UINT#0;   // Внутрішній лічильник циклів без зміни encoder sign-of-life.
      CmdAckError : Bool := FALSE;   // Внутрішній імпульс квітування помилки.
      TempLifeUInt : UInt := UINT#0;   // Тимчасова змінна для виділення encoder sign-of-life.
      TempMasterLifeUInt : UInt := UINT#0;   // Тимчасова змінна для запису master sign-of-life у STW2_ENC.
   END_VAR
   VAR RETAIN
      AckErrorHoldCycles : UInt := UINT#10;   // Кількість циклів утримання STW2_ENC bit 7.
   END_VAR
   VAR
      AckErrorHoldCounter : UInt := UINT#0;   // Поточний лічильник циклів утримання квітування.
   END_VAR
   VAR RETAIN
      PresetTimeoutCycles : UInt := UINT#100;   // Максимальна тривалість очікування preset acknowledgment
   END_VAR
   VAR
      PresetTimeoutCounter : UInt := UINT#0;   // Поточний лічильник очікування
   END_VAR
BEGIN
   //PresetStatus — розшифровка
   //|       Код | Значення                                      |
   //| --------: | --------------------------------------------- |
   //| `16#0000` | Немає помилки.                                |
   //| `16#8201` | `#PresetServiceEnable = FALSE`.                |
   //| `16#8202` | Немає дозволу `PresetPermit`.                 |
   //| `16#8203` | Енкодер не готовий або є помилка комунікації. |
   //| `16#8204` | Preset вже активний.                          |
   //| `16#8205` | `#PresetValueRaw` поза допустимим діапазоном.  |
   //| `16#8206` | Не отримано підтвердження preset протягом заданого часу |


   //Status — діагностичне слово блока
   //| Біт |     Маска | Значення                     |
   //| --: | --------: | ---------------------------- |
   //|   0 | `16#0001` | `#ReadError = TRUE`           |
   //|   1 | `16#0002` | `#WriteError = TRUE`          |
   //|   2 | `16#0004` | `#CommunicationFault = TRUE`  |
   //|   3 | `16#0008` | `#ControlByPlcActive = FALSE` |
   //|   4 | `16#0010` | `#EncoderFault = TRUE`        |
   //|   5 | `16#0020` | `#EncoderAlarm = TRUE`        |
   //|   8 | `16#0100` | `#EncoderLifeValid = FALSE`   |
   //|   9 | `16#0200` | `#PositionDataValid = FALSE`  |
   //|  10 | `16#0400` | `#VelocityDataValid = FALSE`  |
   //|  11 | `16#0800` | `#EncoderReady = FALSE`       |
   //|  12 | `16#1000` | `SimulationActive = TRUE`    |
   //|  13 | `16#2000` | `#PresetBusy = TRUE`          |
   //|  14 | `16#4000` | `#PresetError = TRUE`         |

   // ============================================================
   // 1. Початкові значення на цикл
   // ============================================================

   #Status := W#16#0000;

   #ReadRetVal := INT#0;
   #WriteRetVal := INT#0;

   #ReadError := FALSE;
   #WriteError := FALSE;
   #CommunicationFault := FALSE;

   #PresetAck := FALSE;
   #PositionActualValidBit := FALSE;
   #VelocityActualValidBit := FALSE;
   #EncoderFault := FALSE;
   #EncoderAlarm := FALSE;
   #EncoderErrorCode := DINT#0;
   #ControlByPlcActive := FALSE;

   #PositionDataValid := FALSE;
   #VelocityDataValid := FALSE;
   #EncoderReady := FALSE;

   #EncoderLifeChanged := FALSE;
   #EncoderLifeValid := FALSE;

   #CmdAckError := FALSE;

   #PresetDone := FALSE;
   #PresetAckRising := FALSE;

   #SimulationActive :=
   #SimulationMode
   AND #SimulationPermit;


   // ============================================================
   // 2. Фронти команд
   // ============================================================

   #AckErrorEdge(CLK := #AckError);

   // Load the hold counter on the rising edge.
   IF #AckErrorEdge.Q THEN

       IF #AckErrorHoldCycles = UINT#0 THEN

           // Keep the command for at least one cycle.
           #AckErrorHoldCounter := UINT#1;

       ELSE

           #AckErrorHoldCounter :=
           #AckErrorHoldCycles;

       END_IF;

   END_IF;


   // Keep the acknowledgment command active
   // while the counter is greater than zero.
   #CmdAckError :=
   (#AckErrorHoldCounter > UINT#0);

   #PresetStartEdge(CLK := #PresetStart);


   // ============================================================
   // 3. Читання PZD-даних
   // ============================================================

   IF NOT #Enable THEN

       #ReadError := TRUE;
       #WriteError := TRUE;
       #CommunicationFault := TRUE;

       #PzdInActual.ZSW2_ENC := W#16#0000;
       #PzdInActual.G1_XIST2 := DINT#0;
       #PzdInActual.NIST_B := DINT#0;

   ELSIF #SimulationActive THEN

       IF #SimInputValid THEN

           #PzdInActual := #SimPzdIn;
           #ReadError := FALSE;

       ELSE

           #PzdInActual.ZSW2_ENC := W#16#0000;
           #PzdInActual.G1_XIST2 := DINT#0;
           #PzdInActual.NIST_B := DINT#0;

           #ReadError := TRUE;
           #CommunicationFault := TRUE;

       END_IF;

   ELSE

       #ReadRetVal := DPRD_DAT(
                               LADDR := #HW_ID_Tlg89,
                               RECORD => #PzdIn
       );

       #ReadError :=
       #ReadRetVal <> INT#0;

       IF #ReadError THEN

           #PzdInActual.ZSW2_ENC := W#16#0000;
           #PzdInActual.G1_XIST2 := DINT#0;
           #PzdInActual.NIST_B := DINT#0;

           #CommunicationFault := TRUE;

       ELSE

           #PzdInActual := #PzdIn;

       END_IF;

   END_IF;


   // ============================================================
   // 4. Декодування ZSW2_ENC
   // ============================================================

   // bit 0 = preset acknowledgment
   #PresetAck :=
   (#PzdInActual.ZSW2_ENC AND W#16#0001) <> W#16#0000;

   // bit 1 = position actual value valid
   #PositionActualValidBit :=
   (#PzdInActual.ZSW2_ENC AND W#16#0002) <> W#16#0000;

   // bit 2 = velocity actual value valid
   #VelocityActualValidBit :=
   (#PzdInActual.ZSW2_ENC AND W#16#0004) <> W#16#0000;

   // bit 3 = fault active
   #EncoderFault :=
   (#PzdInActual.ZSW2_ENC AND W#16#0008) <> W#16#0000;

   // During an encoder fault, G1_XIST2 contains the error code.
   IF #EncoderFault THEN

       // Keep only the lower 12 bits.
       #EncoderErrorCode :=
       #PzdInActual.G1_XIST2
       AND DINT#4095;

   ELSE

       #EncoderErrorCode :=
       DINT#0;

   END_IF;


   // bit 7 = alarm / warning
   #EncoderAlarm :=
   (#PzdInActual.ZSW2_ENC AND W#16#0080) <> W#16#0000;

   // bit 9 = control requested / data valid
   #ControlByPlcActive :=
   (#PzdInActual.ZSW2_ENC AND W#16#0200) <> W#16#0000;


   // ============================================================
   // 5. Фронт підтвердження preset
   // ============================================================

   #PresetAckRising :=
   #PresetAck
   AND NOT #PrevPresetAck;

   #PrevPresetAck :=
   #PresetAck;


   // ============================================================
   // 6. Encoder sign-of-life з ZSW2_ENC bits 12...15
   // ============================================================

   #TempLifeUInt :=
   WORD_TO_UINT(#PzdInActual.ZSW2_ENC AND W#16#F000) / UINT#4096;

   #EncoderSignOfLife :=
   UINT_TO_USINT(#TempLifeUInt);

   IF NOT #MonitorSignOfLife THEN

       #EncoderLifeValid := TRUE;
       #EncoderLifeChanged := TRUE;
       #UnchangedLifeCyclesInt := UINT#0;

   ELSE

       IF #EncoderSignOfLife = USINT#0 THEN

           #EncoderLifeValid := FALSE;
           #EncoderLifeChanged := FALSE;

       ELSE

           IF #EncoderSignOfLife <> #LastEncoderLifeCounter THEN

               #EncoderLifeChanged := TRUE;
               #UnchangedLifeCyclesInt := UINT#0;
               #LastEncoderLifeCounter := #EncoderSignOfLife;

           ELSE

               #EncoderLifeChanged := FALSE;

               IF #UnchangedLifeCyclesInt < UINT#65535 THEN
                   #UnchangedLifeCyclesInt :=
                   #UnchangedLifeCyclesInt + UINT#1;
               END_IF;

           END_IF;

           #EncoderLifeValid :=
           #UnchangedLifeCyclesInt <= #MaxUnchangedLifeCycles;

       END_IF;

   END_IF;

   #UnchangedLifeCycles :=
   #UnchangedLifeCyclesInt;


   // ============================================================
   // 7. Достовірність даних Telegram 89
   // ============================================================

   #PositionDataValid :=
   #Enable
   AND NOT #ReadError
   AND #ControlByPlcActive
   AND #PositionActualValidBit
   AND NOT #EncoderFault
   AND
   (
       NOT #MonitorSignOfLife
       OR #EncoderLifeValid
   );

   #VelocityDataValid :=
   #Enable
   AND NOT #ReadError
   AND #ControlByPlcActive
   AND #VelocityActualValidBit
   AND NOT #EncoderFault
   AND
   (
       NOT #MonitorSignOfLife
       OR #EncoderLifeValid
   );


   #CommunicationFault :=
   #CommunicationFault
   OR #ReadError
   OR #WriteError
   OR NOT #ControlByPlcActive
   OR
   (
       #MonitorSignOfLife
       AND NOT #EncoderLifeValid
   );


   // ============================================================
   // 8. Копіювання значень
   // ============================================================

   IF #PositionDataValid THEN
       #AbsolutePositionRaw :=
       #PzdInActual.G1_XIST2;
   END_IF;

   IF #VelocityDataValid THEN
       #VelocityRaw :=
       #PzdInActual.NIST_B;
   ELSE
       #VelocityRaw :=
       DINT#0;
   END_IF;


   // ============================================================
   // 9. Готовність енкодера
   // ============================================================

   #EncoderReady :=
   #Enable
   AND NOT #CommunicationFault
   AND #ControlByPlcActive
   AND #PositionDataValid
   AND #VelocityDataValid
   AND NOT #EncoderFault;


   // ============================================================
   // 10. Preset service
   //
   // Для Telegram 89 preset value передається циклічно
   // через G1_XIST_PRESET_B1.
   // STW2_ENC bit 0 дає фронт запуску preset.
   // ZSW2_ENC bit 0 підтверджує виконання preset.
   // ============================================================

   IF #PresetStartEdge.Q THEN

       IF NOT #PresetServiceEnable THEN

           #PresetError := TRUE;
           #PresetStatus := W#16#8201;

       ELSIF NOT #PresetPermit THEN

           #PresetError := TRUE;
           #PresetStatus := W#16#8202;

       ELSIF NOT #EncoderReady
           OR #CommunicationFault THEN

           #PresetError := TRUE;
           #PresetStatus := W#16#8203;

       ELSIF #PresetBusy THEN

           #PresetError := TRUE;
           #PresetStatus := W#16#8204;

       ELSIF (#PresetValueRaw < DINT#0)
           OR (#PresetValueRaw > #MaxPositionRaw) THEN

           #PresetError := TRUE;
           #PresetStatus := W#16#8205;

       ELSE

           // Запускаємо preset.
           // Bit 0 у STW2_ENC буде встановлений, поки не прийде ack.
           #PresetBusy := TRUE;
           #PresetError := FALSE;
           #PresetStatus := W#16#0000;

           #ActivePresetValueRaw :=
           #PresetValueRaw;

           // Reset preset timeout counter.
           #PresetTimeoutCounter := UINT#0;

       END_IF;

   END_IF;

   // Successful preset acknowledgment.
   IF #PresetBusy
       AND #PresetAckRising THEN

       #PresetBusy := FALSE;
       #PresetDone := TRUE;
       #PresetStatus := W#16#0000;

   END_IF;

   // ============================================================
   // Preset timeout monitoring
   // ============================================================
   // Timeout is checked only if preset is still busy.
   IF #PresetBusy THEN

       IF #PresetTimeoutCounter < UINT#65535 THEN

           #PresetTimeoutCounter :=
           #PresetTimeoutCounter + UINT#1;

       END_IF;


       IF #PresetTimeoutCounter >= #PresetTimeoutCycles THEN

           #PresetBusy := FALSE;
           #PresetError := TRUE;
           #PresetStatus := W#16#8206;

       END_IF;

   ELSE

       #PresetTimeoutCounter := UINT#0;

   END_IF;

   // ============================================================
   // 11. Формування STW2_ENC та G1_XIST_PRESET_B1
   // ============================================================

   #PzdOut.STW2_ENC := W#16#0000;
   #PzdOut.G1_XIST_PRESET_B1 := DINT#0;

   // STW2_ENC bit 0 = XIST_PRESET_CONTROL.
   // Rising edge запускає preset.
   IF #PresetBusy
       AND #Enable THEN

       #PzdOut.STW2_ENC :=
       #PzdOut.STW2_ENC OR W#16#0001;

       #PzdOut.G1_XIST_PRESET_B1 :=
       #ActivePresetValueRaw;

   END_IF;

   // STW2_ENC bit 7 = acknowledge error.
   IF #CmdAckError
       AND #Enable THEN

       #PzdOut.STW2_ENC :=
       #PzdOut.STW2_ENC OR W#16#0080;

   END_IF;

   // STW2_ENC bit 10 = check by control / cyclic data valid.
   IF #Enable THEN

       #PzdOut.STW2_ENC :=
       #PzdOut.STW2_ENC OR W#16#0400;

   END_IF;

   // STW2_ENC bits 12...15 = master sign-of-life.
   IF #EnableSignOfLife
       AND #Enable THEN

       #MasterSignOfLife :=
       #MasterLifeCounter;

       #TempMasterLifeUInt :=
       USINT_TO_UINT(#MasterLifeCounter) * UINT#4096;

       #PzdOut.STW2_ENC :=
       (#PzdOut.STW2_ENC AND W#16#0FFF)
       OR UINT_TO_WORD(#TempMasterLifeUInt);

       IF #MasterLifeCounter >= USINT#15 THEN
           #MasterLifeCounter := USINT#1;
       ELSE
           #MasterLifeCounter :=
           #MasterLifeCounter + USINT#1;
       END_IF;

   ELSE

       #MasterSignOfLife := USINT#0;

   END_IF;

   #PzdOutActual :=
   #PzdOut;

   #SimPzdOut :=
   #PzdOut;

   // Decrease the acknowledgment hold counter
   // after the telegram was copied to all outputs.
   IF #AckErrorHoldCounter > UINT#0 THEN

       #AckErrorHoldCounter :=
       #AckErrorHoldCounter - UINT#1;

   END_IF;

   // ============================================================
   // 12. Запис PZD-даних
   // ============================================================

   IF NOT #Enable THEN

       #WriteError := TRUE;
       #CommunicationFault := TRUE;

   ELSIF #SimulationActive THEN

       #WriteError := FALSE;

   ELSE

       #WriteRetVal := DPWR_DAT(
                                LADDR := #HW_ID_Tlg89,
                                RECORD := #PzdOut
       );

       #WriteError :=
       #WriteRetVal <> INT#0;

       IF #WriteError THEN
           #CommunicationFault := TRUE;
       END_IF;

   END_IF;


   // ============================================================
   // 13. Уточнення після запису
   // ============================================================

   IF #WriteError THEN
       #EncoderReady := FALSE;
       #PositionDataValid := FALSE;
       #VelocityDataValid := FALSE;
   END_IF;


   // ============================================================
   // 14. Діагностичне слово
   // ============================================================

   IF #ReadError THEN
       #Status := #Status OR W#16#0001;
   END_IF;

   IF #WriteError THEN
       #Status := #Status OR W#16#0002;
   END_IF;

   IF #CommunicationFault THEN
       #Status := #Status OR W#16#0004;
   END_IF;

   IF NOT #ControlByPlcActive THEN
       #Status := #Status OR W#16#0008;
   END_IF;

   IF #EncoderFault THEN
       #Status := #Status OR W#16#0010;
   END_IF;

   IF #EncoderAlarm THEN
       #Status := #Status OR W#16#0020;
   END_IF;

   IF  #MonitorSignOfLife AND NOT #EncoderLifeValid THEN
       #Status := #Status OR W#16#0100;
   END_IF;

   IF NOT #PositionDataValid THEN
       #Status := #Status OR W#16#0200;
   END_IF;

   IF NOT #VelocityDataValid THEN
       #Status := #Status OR W#16#0400;
   END_IF;

   IF NOT #EncoderReady THEN
       #Status := #Status OR W#16#0800;
   END_IF;

   IF #SimulationActive THEN
       #Status := #Status OR W#16#1000;
   END_IF;

   IF #PresetBusy THEN
       #Status := #Status OR W#16#2000;
   END_IF;

   IF #PresetError THEN
       #Status := #Status OR W#16#4000;
   END_IF;
END_FUNCTION_BLOCK

FUNCTION_BLOCK "FB_PositionCorrection"   // FB82, LAD
{ S7_Optimized_Access := 'TRUE' }
VERSION : 0.1
   VAR_INPUT
      ix_Enable : Bool := FALSE;   // Загальний дозвіл роботи блока корекції координати.
      il_PositionScaled_mm : LReal := 0.0;   // Поточна координата після FC_EncoderScale, до програмної корекції.
      ix_PositionValid : Bool := FALSE;   // TRUE — вхідна масштабована координата достовірна.
      ix_ReferenceSwitch : Bool := FALSE;   // Сигнал реперного шляхового вимикача. TRUE — вимикач не натиснутий; FALSE — механізм наїхав на вимикач.
      il_ReferencePosition_mm : LReal := 0.0;   // Жорстко задана координата реперної точки, мм.
      il_VirtualOffset_mm : LReal := 0.0;   // Пусконалагоджувальне віртуальне зміщення реперної координати, мм.
      ix_AutoCorrectionEnable : Bool := TRUE;   // Дозвіл фонової автоматичної корекції по реперному вимикачу.
      ix_CalibrationActive : Bool := FALSE;   // TRUE — виконується повна процедура калібрування; фонова корекція блокується.
      ix_CalibrationCompleted : Bool := FALSE;   // Ознака успішно завершеної повної калібровки. По передньому фронту програмна корекція обнуляється.
   END_VAR
   VAR_OUTPUT
      ql_PositionCorrected_mm : LReal := 0.0;   // Робоча скоригована координата механізму, мм.
      qd_PositionCorrectedRounded_mm : DInt := 0;   // Скоригована координата, округлена до цілого мм.
      ql_CorrectionOffset_mm : LReal := 0.0;   // Поточна програмна поправка координати.
      qx_CorrectionValid : Bool := FALSE;   // TRUE — програмна корекція має валідний стан.
      qx_AutoCorrectionDone : Bool := FALSE;   // Одноцикловий імпульс успішної фонової автокорекції.
      qx_ReferenceFalling : Bool := FALSE;   // Одноцикловий імпульс спадного фронту реперного вимикача.
      ql_LastCorrectionDelta_mm : LReal := 0.0;   // Величина останньої виконаної автокорекції, мм.
      qw_Status : Word := W#16#0000;   // Діагностичне слово блока.
   END_VAR
   VAR
      stat_ReferenceOld : Bool := FALSE;   // Попередній стан реперного вимикача для визначення спадного фронту.
      stat_CalibrationCompletedOld : Bool := FALSE;   // Попередній стан ознаки завершення калібровки.
   END_VAR
   VAR RETAIN
      stat_CorrectionOffset_mm : LReal := 0.0;   // Збережена програмна поправка координати.
      stat_CorrectionValid : Bool := FALSE;   // Збережена ознака валідності програмної поправки.
   END_VAR
   VAR
      stat_LastCorrectionDelta_mm : LReal := 0.0;   // Величина останньої виконаної автокорекції.
   END_VAR
   VAR_TEMP
      ReferenceFalling : Bool;   // Спадний фронт реперного вимикача.
      CalibrationCompletedEdge : Bool;   // Передній фронт успішного завершення калібровки.
      ReferenceTarget_mm : LReal;   // Правильна координата в точці спрацювання репера.
      NewCorrectionOffset_mm : LReal;   // Нове розраховане накопичене зміщення.
   END_VAR
BEGIN

REGION Network 1 (SCL): Спадний фронт реперного вимикача.
   // ============================================================
   // FB_PositionCorrection
   //
   // Фонова програмна корекція координати механізму.
   //
   // Вхідна координата надходить після FC_EncoderScale.
   //
   // Під час нормальної роботи нове зміщення розраховується
   // по спадному фронту реперного шляхового вимикача.
   //
   // Під час повної калібровки фонова корекція заблокована.
   //
   // Після успішної повної калібровки програмне зміщення
   // обнуляється, оскільки правильна система координат уже
   // встановлена апаратним preset енкодера.
   // ============================================================


   // ============================================================
   // 1. Формування фронтів
   // ============================================================

   // Реперний вимикач:
   // TRUE  - механізм ще не наїхав на вимикач.
   // FALSE - механізм наїхав на вимикач.
   //
   // Реперна точка визначається переходом TRUE -> FALSE.

   #ReferenceFalling :=
   #stat_ReferenceOld
   AND NOT #ix_ReferenceSwitch;

   #qx_ReferenceFalling :=
   #ReferenceFalling;


   // Передній фронт успішного завершення повної калібровки.

   #CalibrationCompletedEdge :=
   #ix_CalibrationCompleted
   AND NOT #stat_CalibrationCompletedOld;


   // ============================================================
   // 2. Початкові значення одноциклових виходів
   // ============================================================

   #qx_AutoCorrectionDone := FALSE;


   // ============================================================
   // 3. Обробка успішного завершення повної калібровки
   // ============================================================

   // Після успішного hardware preset масштабована координата
   // вже знаходиться у правильній системі координат.
   //
   // Тому додаткове програмне зміщення більше не потрібне.
   //
   // Ця операція має вищий пріоритет за фонову автокорекцію.

   IF #CalibrationCompletedEdge THEN

       #stat_CorrectionOffset_mm := 0.0;

       #stat_CorrectionValid := TRUE;

       #stat_LastCorrectionDelta_mm := 0.0;


       // ============================================================
       // 4. Фонова автоматична корекція координати
       // ============================================================

       // Корекція виконується тільки:
       // - якщо блок увімкнений;
       // - якщо фонова корекція дозволена;
       // - якщо поточна координата достовірна;
       // - якщо повна калібровка не активна;
       // - у момент спадного фронту реперного вимикача.

   ELSIF #ix_Enable
       AND #ix_AutoCorrectionEnable
       AND #ix_PositionValid
       AND NOT #ix_CalibrationActive
       AND #ReferenceFalling
   THEN

       // Правильна координата механізму
       // в момент спрацювання реперного вимикача.
       //
       // Віртуальне зміщення задається під час ПНР.

       #ReferenceTarget_mm :=
       #il_ReferencePosition_mm
       + #il_VirtualOffset_mm;


       // Розрахунок нового повного програмного зміщення.
       //
       // Після розрахунку повинно виконуватися:
       //
       // PositionScaled_mm + CorrectionOffset_mm
       // =
       // ReferencePosition_mm + VirtualOffset_mm

       #NewCorrectionOffset_mm :=
       #ReferenceTarget_mm
       - #il_PositionScaled_mm;


       // Визначаємо, наскільки фактично змінилася
       // робоча координата при цій автокорекції.
       //
       // Наприклад:
       // старий offset = +2.0 мм
       // новий offset  = +3.5 мм
       //
       // LastCorrectionDelta = +1.5 мм

       #stat_LastCorrectionDelta_mm :=
       #NewCorrectionOffset_mm
       - #stat_CorrectionOffset_mm;


       // Запам'ятовуємо нове повне зміщення.

       #stat_CorrectionOffset_mm :=
       #NewCorrectionOffset_mm;


       // Зміщення тепер має валідне значення.

       #stat_CorrectionValid := TRUE;


       // Одноцикловий імпульс успішної автокорекції.

       #qx_AutoCorrectionDone := TRUE;

   END_IF;


   // ============================================================
   // 5. Формування скоригованої координати
   // ============================================================

   // Якщо програмне зміщення вже валідне,
   // використовуємо його.
   //
   // Якщо корекція ще жодного разу не була встановлена,
   // передаємо масштабовану координату без змін.

   IF #stat_CorrectionValid THEN

       #ql_PositionCorrected_mm :=
       #il_PositionScaled_mm
       + #stat_CorrectionOffset_mm;

   ELSE

       #ql_PositionCorrected_mm :=
       #il_PositionScaled_mm;

   END_IF;


   // Округлена робоча координата.

   #qd_PositionCorrectedRounded_mm :=
   LREAL_TO_DINT(#ql_PositionCorrected_mm);


   // ============================================================
   // 6. Формування виходів стану корекції
   // ============================================================

   #ql_CorrectionOffset_mm :=
   #stat_CorrectionOffset_mm;

   #qx_CorrectionValid :=
   #stat_CorrectionValid;

   #ql_LastCorrectionDelta_mm :=
   #stat_LastCorrectionDelta_mm;


   // ============================================================
   // 7. Діагностичне слово
   //
   // Bit 0 - блок увімкнений
   // Bit 1 - масштабована координата достовірна
   // Bit 2 - програмна корекція валідна
   // Bit 3 - фонова автокорекція дозволена
   // Bit 4 - активна повна калібровка
   // Bit 5 - виявлено спадний фронт репера
   // Bit 6 - у цьому циклі виконана автокорекція
   // ============================================================

   #qw_Status := W#16#0000;


   // Bit 0 - блок увімкнений.

   IF #ix_Enable THEN

       #qw_Status :=
       #qw_Status OR W#16#0001;

   END_IF;


   // Bit 1 - вхідна координата достовірна.

   IF #ix_PositionValid THEN

       #qw_Status :=
       #qw_Status OR W#16#0002;

   END_IF;


   // Bit 2 - програмна корекція валідна.

   IF #stat_CorrectionValid THEN

       #qw_Status :=
       #qw_Status OR W#16#0004;

   END_IF;


   // Bit 3 - фонова автокорекція дозволена.

   IF #ix_AutoCorrectionEnable THEN

       #qw_Status :=
       #qw_Status OR W#16#0008;

   END_IF;


   // Bit 4 - активна процедура повної калібровки.

   IF #ix_CalibrationActive THEN

       #qw_Status :=
       #qw_Status OR W#16#0010;

   END_IF;


   // Bit 5 - спадний фронт реперного вимикача.

   IF #ReferenceFalling THEN

       #qw_Status :=
       #qw_Status OR W#16#0020;

   END_IF;


   // Bit 6 - автокорекція виконана у цьому циклі.

   IF #qx_AutoCorrectionDone THEN

       #qw_Status :=
       #qw_Status OR W#16#0040;

   END_IF;


   // ============================================================
   // 8. Запам'ятовування станів для наступного циклу PLC
   // ============================================================

   #stat_ReferenceOld :=
   #ix_ReferenceSwitch;

   #stat_CalibrationCompletedOld :=
   #ix_CalibrationCompleted;
END_REGION
END_FUNCTION_BLOCK

FUNCTION "FC_Enc_Pos_Call" : Void   // FC80, LAD
TITLE = Енкодери та позиціонування механізмів крана
{ S7_Optimized_Access := 'TRUE' }
VERSION : 0.1
   VAR_TEMP
      "1BR_Config_Valid" : Bool;
      "3BR_Config_Valid" : Bool;
      "4BR1_Config_Valid" : Bool;
      "4BR2_Config_Valid" : Bool;
   END_VAR
   VAR_TEMP   // added for the SCL form of the ladder/FBD networks
      _w1 : Bool;
      _w2 : Bool;
   END_VAR
BEGIN

REGION Network 2 (SCL): ====== Підйом (Lifting/Hoist) ======
END_REGION

REGION Network 3: Зв'язок з енкодером підйому 1BR
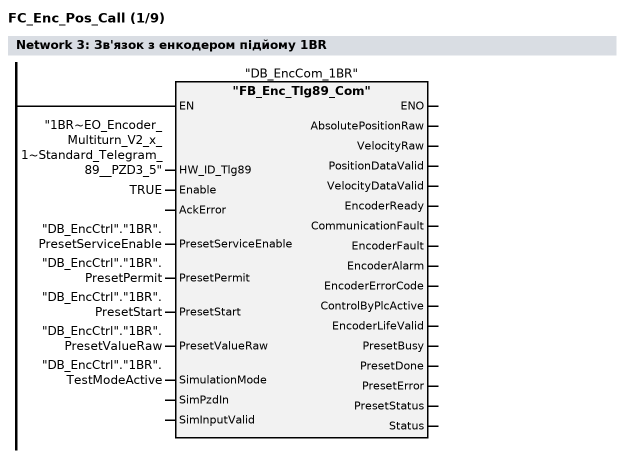
   RUNG wire#powerrail
      "DB_EncCom_1BR"(HW_ID_Tlg89 := "1BR~EO_Encoder_Multiturn_V2_x_1~Standard_Telegram_89__PZD3_5", Enable := TRUE, AckError :=, PresetServiceEnable := "DB_EncCtrl"."1BR".PresetServiceEnable, PresetPermit := "DB_EncCtrl"."1BR".PresetPermit, PresetStart := "DB_EncCtrl"."1BR".PresetStart, PresetValueRaw := "DB_EncCtrl"."1BR".PresetValueRaw, SimulationMode := "DB_EncCtrl"."1BR".TestModeActive, SimPzdIn :=, SimInputValid :=, AbsolutePositionRaw =>, VelocityRaw =>, PositionDataValid =>, VelocityDataValid =>, EncoderReady =>, CommunicationFault =>, EncoderFault =>, EncoderAlarm =>, EncoderErrorCode =>, ControlByPlcActive =>, EncoderLifeValid =>, PresetBusy =>, PresetDone =>, PresetError =>, PresetStatus =>, Status =>)
   END_RUNG
   // the same network as SCL:
   "DB_EncCom_1BR"(HW_ID_Tlg89 := "1BR~EO_Encoder_Multiturn_V2_x_1~Standard_Telegram_89__PZD3_5",   // "FB_Enc_Tlg89_Com"
                   Enable := TRUE,
                   PresetServiceEnable := "DB_EncCtrl"."1BR".PresetServiceEnable,
                   PresetPermit := "DB_EncCtrl"."1BR".PresetPermit,
                   PresetStart := "DB_EncCtrl"."1BR".PresetStart,
                   PresetValueRaw := "DB_EncCtrl"."1BR".PresetValueRaw,
                   SimulationMode := "DB_EncCtrl"."1BR".TestModeActive);
END_REGION

REGION Network 4: Масштабування положення екнодеру підйому 1BR
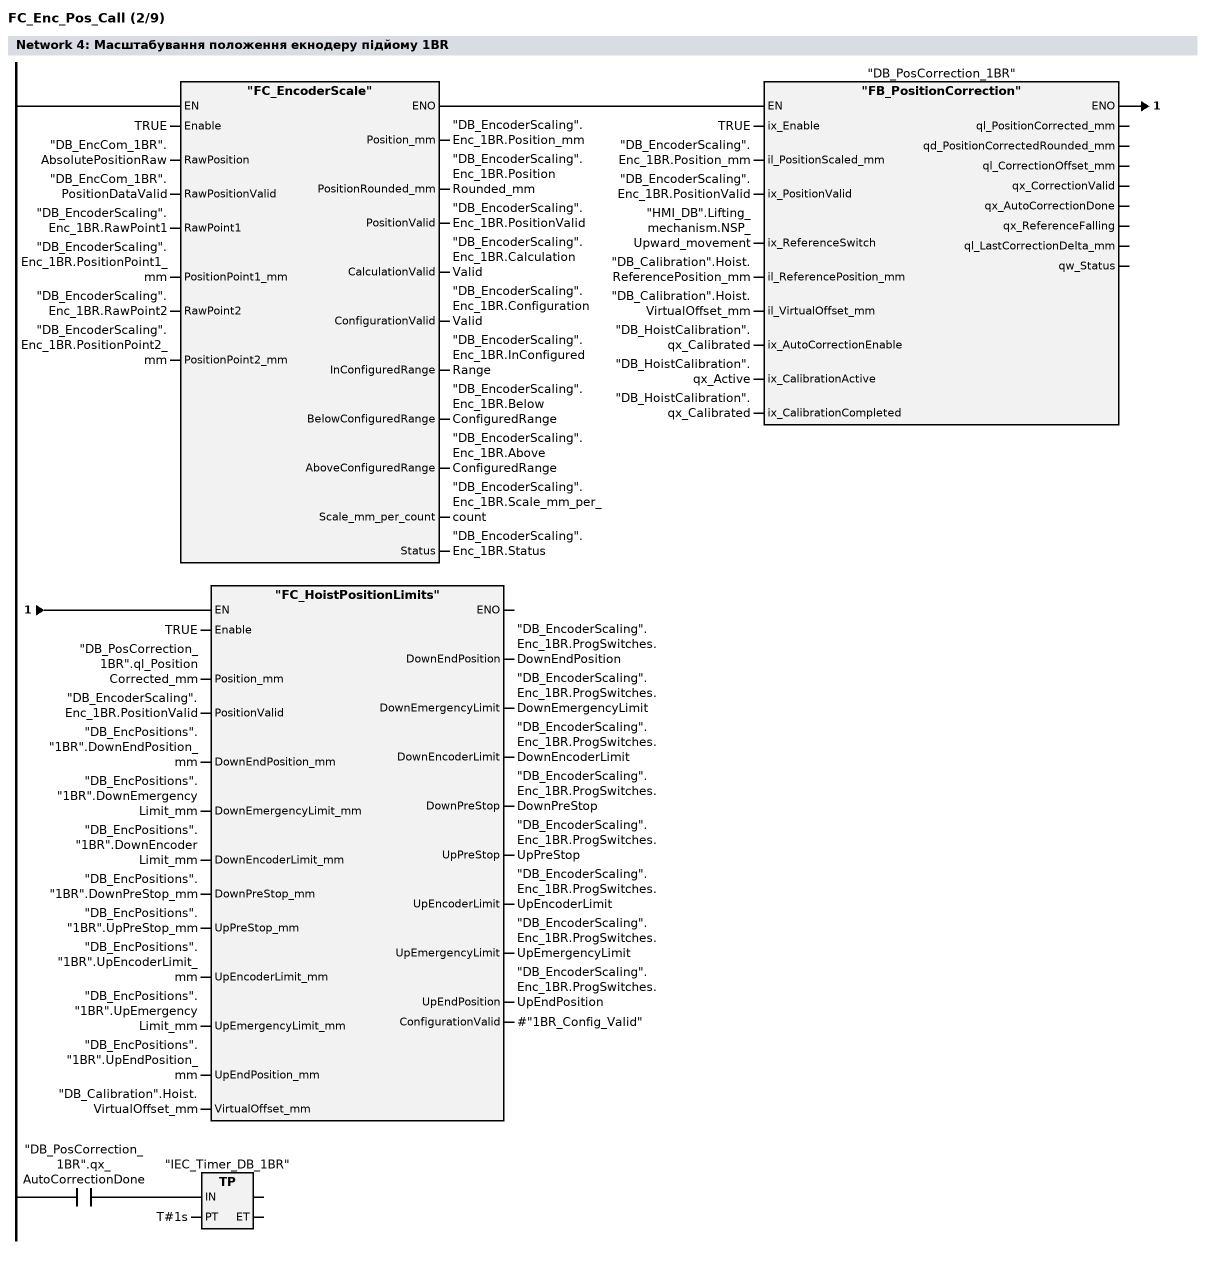
   "FC_EncoderScale"(Enable := TRUE,
                     RawPosition := "DB_EncCom_1BR".AbsolutePositionRaw,
                     RawPositionValid := "DB_EncCom_1BR".PositionDataValid,
                     RawPoint1 := "DB_EncoderScaling".Enc_1BR.RawPoint1,
                     PositionPoint1_mm := "DB_EncoderScaling".Enc_1BR.PositionPoint1_mm,
                     RawPoint2 := "DB_EncoderScaling".Enc_1BR.RawPoint2,
                     PositionPoint2_mm := "DB_EncoderScaling".Enc_1BR.PositionPoint2_mm,
                     Position_mm => "DB_EncoderScaling".Enc_1BR.Position_mm,
                     PositionRounded_mm => "DB_EncoderScaling".Enc_1BR.PositionRounded_mm,
                     PositionValid => "DB_EncoderScaling".Enc_1BR.PositionValid,
                     CalculationValid => "DB_EncoderScaling".Enc_1BR.CalculationValid,
                     ConfigurationValid => "DB_EncoderScaling".Enc_1BR.ConfigurationValid,
                     InConfiguredRange => "DB_EncoderScaling".Enc_1BR.InConfiguredRange,
                     BelowConfiguredRange => "DB_EncoderScaling".Enc_1BR.BelowConfiguredRange,
                     AboveConfiguredRange => "DB_EncoderScaling".Enc_1BR.AboveConfiguredRange,
                     Scale_mm_per_count => "DB_EncoderScaling".Enc_1BR.Scale_mm_per_count,
                     Status => "DB_EncoderScaling".Enc_1BR.Status,
                     ENO => #_w1);
   "DB_PosCorrection_1BR"(EN := #_w1,   // "FB_PositionCorrection"
                          ix_Enable := TRUE,
                          il_PositionScaled_mm := "DB_EncoderScaling".Enc_1BR.Position_mm,
                          ix_PositionValid := "DB_EncoderScaling".Enc_1BR.PositionValid,
                          ix_ReferenceSwitch := "HMI_DB".Lifting_mechanism.NSP_Upward_movement,
                          il_ReferencePosition_mm := "DB_Calibration".Hoist.ReferencePosition_mm,
                          il_VirtualOffset_mm := "DB_Calibration".Hoist.VirtualOffset_mm,
                          ix_AutoCorrectionEnable := "DB_HoistCalibration".qx_Calibrated,
                          ix_CalibrationActive := "DB_HoistCalibration".qx_Active,
                          ix_CalibrationCompleted := "DB_HoistCalibration".qx_Calibrated,
                          ENO => #_w2);
   IF #_w2 THEN
       "FC_HoistPositionLimits"(Enable := TRUE,
                               Position_mm := "DB_PosCorrection_1BR".ql_PositionCorrected_mm,
                               PositionValid := "DB_EncoderScaling".Enc_1BR.PositionValid,
                               DownEndPosition_mm := "DB_EncPositions"."1BR".DownEndPosition_mm,
                               DownEmergencyLimit_mm := "DB_EncPositions"."1BR".DownEmergencyLimit_mm,
                               DownEncoderLimit_mm := "DB_EncPositions"."1BR".DownEncoderLimit_mm,
                               DownPreStop_mm := "DB_EncPositions"."1BR".DownPreStop_mm,
                               UpPreStop_mm := "DB_EncPositions"."1BR".UpPreStop_mm,
                               UpEncoderLimit_mm := "DB_EncPositions"."1BR".UpEncoderLimit_mm,
                               UpEmergencyLimit_mm := "DB_EncPositions"."1BR".UpEmergencyLimit_mm,
                               UpEndPosition_mm := "DB_EncPositions"."1BR".UpEndPosition_mm,
                               VirtualOffset_mm := "DB_Calibration".Hoist.VirtualOffset_mm,
                               DownEndPosition => "DB_EncoderScaling".Enc_1BR.ProgSwitches.DownEndPosition,
                               DownEmergencyLimit => "DB_EncoderScaling".Enc_1BR.ProgSwitches.DownEmergencyLimit,
                               DownEncoderLimit => "DB_EncoderScaling".Enc_1BR.ProgSwitches.DownEncoderLimit,
                               DownPreStop => "DB_EncoderScaling".Enc_1BR.ProgSwitches.DownPreStop,
                               UpPreStop => "DB_EncoderScaling".Enc_1BR.ProgSwitches.UpPreStop,
                               UpEncoderLimit => "DB_EncoderScaling".Enc_1BR.ProgSwitches.UpEncoderLimit,
                               UpEmergencyLimit => "DB_EncoderScaling".Enc_1BR.ProgSwitches.UpEmergencyLimit,
                               UpEndPosition => "DB_EncoderScaling".Enc_1BR.ProgSwitches.UpEndPosition,
                               ConfigurationValid => #"1BR_Config_Valid");
   END_IF;
   "IEC_Timer_DB_1BR".TP(IN := "DB_PosCorrection_1BR".qx_AutoCorrectionDone, PT := T#1s);
END_REGION

REGION Network 6 (SCL): ====== Пересування візка (Trolley_movement) ======
END_REGION

REGION Network 7: Зв'язок з енкодером візка 3BR
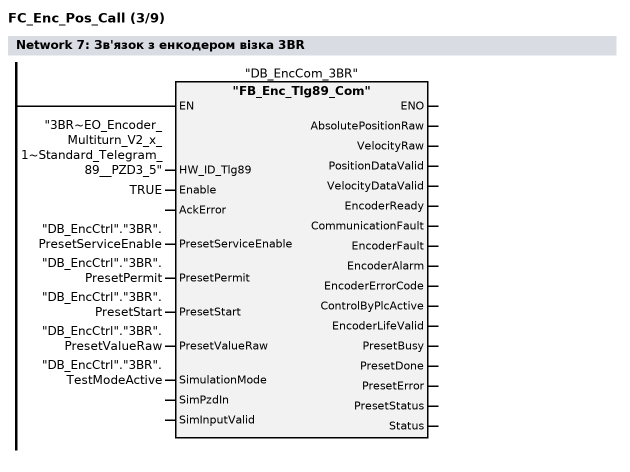
   RUNG wire#powerrail
      "DB_EncCom_3BR"(HW_ID_Tlg89 := "3BR~EO_Encoder_Multiturn_V2_x_1~Standard_Telegram_89__PZD3_5", Enable := TRUE, AckError :=, PresetServiceEnable := "DB_EncCtrl"."3BR".PresetServiceEnable, PresetPermit := "DB_EncCtrl"."3BR".PresetPermit, PresetStart := "DB_EncCtrl"."3BR".PresetStart, PresetValueRaw := "DB_EncCtrl"."3BR".PresetValueRaw, SimulationMode := "DB_EncCtrl"."3BR".TestModeActive, SimPzdIn :=, SimInputValid :=, AbsolutePositionRaw =>, VelocityRaw =>, PositionDataValid =>, VelocityDataValid =>, EncoderReady =>, CommunicationFault =>, EncoderFault =>, EncoderAlarm =>, EncoderErrorCode =>, ControlByPlcActive =>, EncoderLifeValid =>, PresetBusy =>, PresetDone =>, PresetError =>, PresetStatus =>, Status =>)
   END_RUNG
   // the same network as SCL:
   "DB_EncCom_3BR"(HW_ID_Tlg89 := "3BR~EO_Encoder_Multiturn_V2_x_1~Standard_Telegram_89__PZD3_5",   // "FB_Enc_Tlg89_Com"
                   Enable := TRUE,
                   PresetServiceEnable := "DB_EncCtrl"."3BR".PresetServiceEnable,
                   PresetPermit := "DB_EncCtrl"."3BR".PresetPermit,
                   PresetStart := "DB_EncCtrl"."3BR".PresetStart,
                   PresetValueRaw := "DB_EncCtrl"."3BR".PresetValueRaw,
                   SimulationMode := "DB_EncCtrl"."3BR".TestModeActive);
END_REGION

REGION Network 8: Масштабування положення енкодера візка 3BR / Масштабування положення екнодеру підйому 1BR
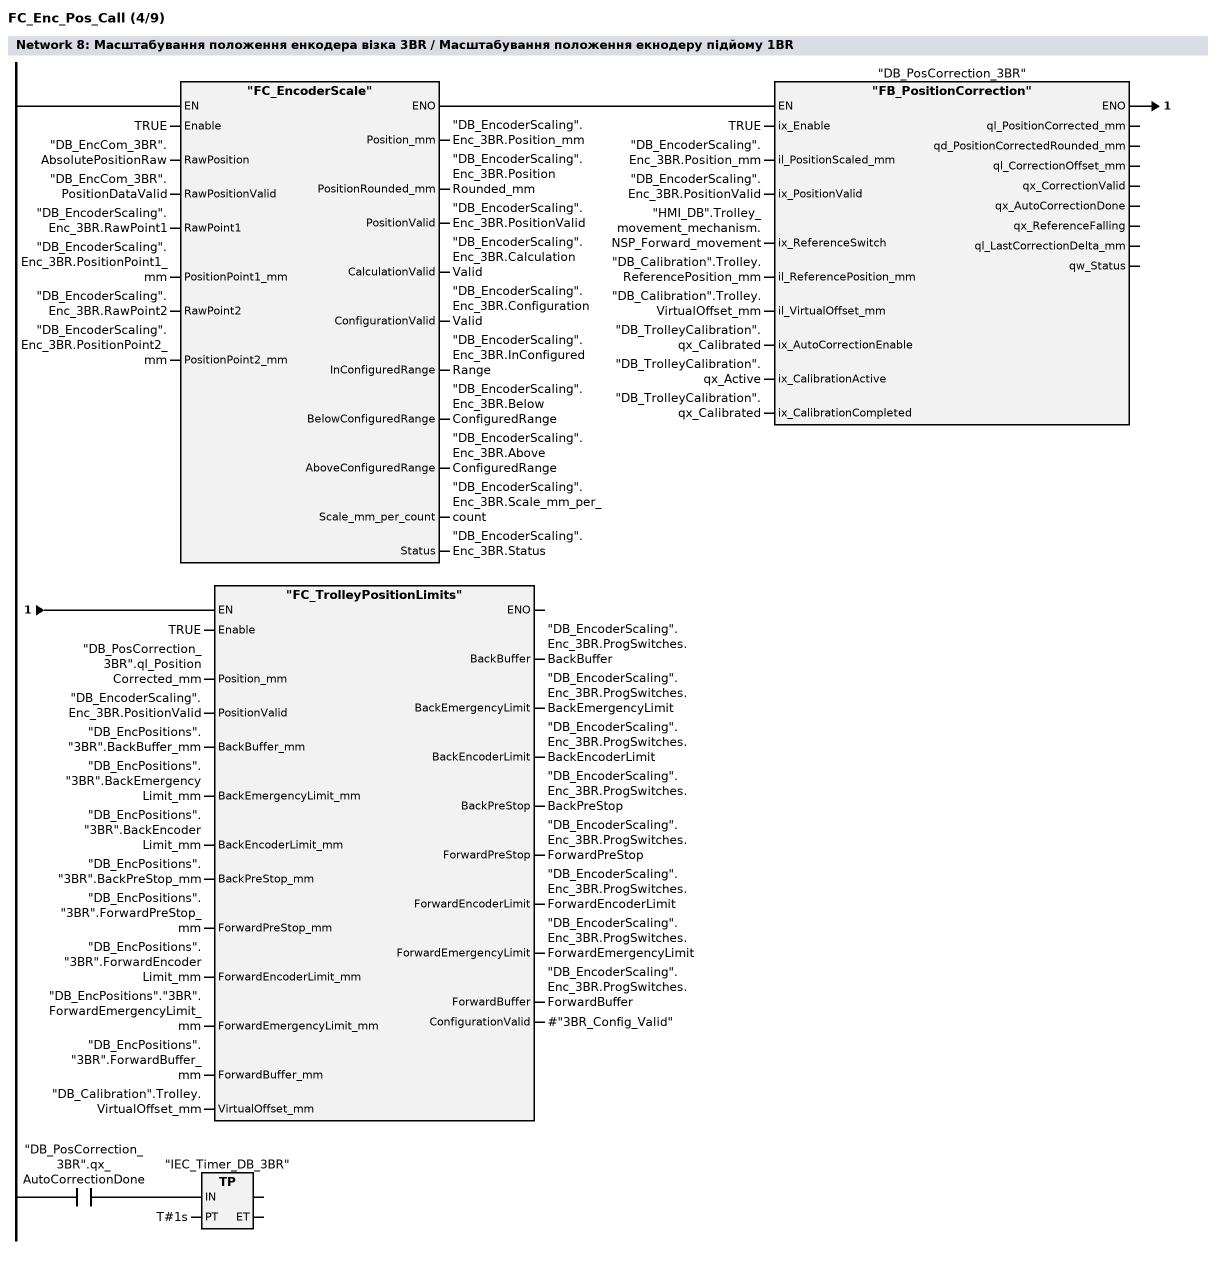
   "FC_EncoderScale"(Enable := TRUE,
                     RawPosition := "DB_EncCom_3BR".AbsolutePositionRaw,
                     RawPositionValid := "DB_EncCom_3BR".PositionDataValid,
                     RawPoint1 := "DB_EncoderScaling".Enc_3BR.RawPoint1,
                     PositionPoint1_mm := "DB_EncoderScaling".Enc_3BR.PositionPoint1_mm,
                     RawPoint2 := "DB_EncoderScaling".Enc_3BR.RawPoint2,
                     PositionPoint2_mm := "DB_EncoderScaling".Enc_3BR.PositionPoint2_mm,
                     Position_mm => "DB_EncoderScaling".Enc_3BR.Position_mm,
                     PositionRounded_mm => "DB_EncoderScaling".Enc_3BR.PositionRounded_mm,
                     PositionValid => "DB_EncoderScaling".Enc_3BR.PositionValid,
                     CalculationValid => "DB_EncoderScaling".Enc_3BR.CalculationValid,
                     ConfigurationValid => "DB_EncoderScaling".Enc_3BR.ConfigurationValid,
                     InConfiguredRange => "DB_EncoderScaling".Enc_3BR.InConfiguredRange,
                     BelowConfiguredRange => "DB_EncoderScaling".Enc_3BR.BelowConfiguredRange,
                     AboveConfiguredRange => "DB_EncoderScaling".Enc_3BR.AboveConfiguredRange,
                     Scale_mm_per_count => "DB_EncoderScaling".Enc_3BR.Scale_mm_per_count,
                     Status => "DB_EncoderScaling".Enc_3BR.Status,
                     ENO => #_w1);
   "DB_PosCorrection_3BR"(EN := #_w1,   // "FB_PositionCorrection"
                          ix_Enable := TRUE,
                          il_PositionScaled_mm := "DB_EncoderScaling".Enc_3BR.Position_mm,
                          ix_PositionValid := "DB_EncoderScaling".Enc_3BR.PositionValid,
                          ix_ReferenceSwitch := "HMI_DB".Trolley_movement_mechanism.NSP_Forward_movement,
                          il_ReferencePosition_mm := "DB_Calibration".Trolley.ReferencePosition_mm,
                          il_VirtualOffset_mm := "DB_Calibration".Trolley.VirtualOffset_mm,
                          ix_AutoCorrectionEnable := "DB_TrolleyCalibration".qx_Calibrated,
                          ix_CalibrationActive := "DB_TrolleyCalibration".qx_Active,
                          ix_CalibrationCompleted := "DB_TrolleyCalibration".qx_Calibrated,
                          ENO => #_w2);
   IF #_w2 THEN
       "FC_TrolleyPositionLimits"(Enable := TRUE,
                               Position_mm := "DB_PosCorrection_3BR".ql_PositionCorrected_mm,
                               PositionValid := "DB_EncoderScaling".Enc_3BR.PositionValid,
                               BackBuffer_mm := "DB_EncPositions"."3BR".BackBuffer_mm,
                               BackEmergencyLimit_mm := "DB_EncPositions"."3BR".BackEmergencyLimit_mm,
                               BackEncoderLimit_mm := "DB_EncPositions"."3BR".BackEncoderLimit_mm,
                               BackPreStop_mm := "DB_EncPositions"."3BR".BackPreStop_mm,
                               ForwardPreStop_mm := "DB_EncPositions"."3BR".ForwardPreStop_mm,
                               ForwardEncoderLimit_mm := "DB_EncPositions"."3BR".ForwardEncoderLimit_mm,
                               ForwardEmergencyLimit_mm := "DB_EncPositions"."3BR".ForwardEmergencyLimit_mm,
                               ForwardBuffer_mm := "DB_EncPositions"."3BR".ForwardBuffer_mm,
                               VirtualOffset_mm := "DB_Calibration".Trolley.VirtualOffset_mm,
                               BackBuffer => "DB_EncoderScaling".Enc_3BR.ProgSwitches.BackBuffer,
                               BackEmergencyLimit => "DB_EncoderScaling".Enc_3BR.ProgSwitches.BackEmergencyLimit,
                               BackEncoderLimit => "DB_EncoderScaling".Enc_3BR.ProgSwitches.BackEncoderLimit,
                               BackPreStop => "DB_EncoderScaling".Enc_3BR.ProgSwitches.BackPreStop,
                               ForwardPreStop => "DB_EncoderScaling".Enc_3BR.ProgSwitches.ForwardPreStop,
                               ForwardEncoderLimit => "DB_EncoderScaling".Enc_3BR.ProgSwitches.ForwardEncoderLimit,
                               ForwardEmergencyLimit => "DB_EncoderScaling".Enc_3BR.ProgSwitches.ForwardEmergencyLimit,
                               ForwardBuffer => "DB_EncoderScaling".Enc_3BR.ProgSwitches.ForwardBuffer,
                               ConfigurationValid => #"3BR_Config_Valid");
   END_IF;
   "IEC_Timer_DB_3BR".TP(IN := "DB_PosCorrection_3BR".qx_AutoCorrectionDone, PT := T#1s);
END_REGION

REGION Network 10 (SCL): ====== Пересування крана - енкодер #1 (Bridge/Crane movement - encoder #1) ====== / ====== Пересування крана - енкодер #1 (Crane movement - encoder #1) ======
END_REGION

REGION Network 11: Зв'язок з енкодером #1 крана 4BR1
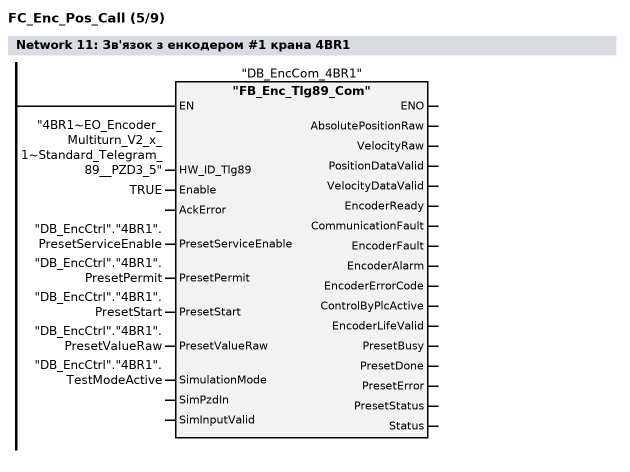
   RUNG wire#powerrail
      "DB_EncCom_4BR1"(HW_ID_Tlg89 := "4BR1~EO_Encoder_Multiturn_V2_x_1~Standard_Telegram_89__PZD3_5", Enable := TRUE, AckError :=, PresetServiceEnable := "DB_EncCtrl"."4BR1".PresetServiceEnable, PresetPermit := "DB_EncCtrl"."4BR1".PresetPermit, PresetStart := "DB_EncCtrl"."4BR1".PresetStart, PresetValueRaw := "DB_EncCtrl"."4BR1".PresetValueRaw, SimulationMode := "DB_EncCtrl"."4BR1".TestModeActive, SimPzdIn :=, SimInputValid :=, AbsolutePositionRaw =>, VelocityRaw =>, PositionDataValid =>, VelocityDataValid =>, EncoderReady =>, CommunicationFault =>, EncoderFault =>, EncoderAlarm =>, EncoderErrorCode =>, ControlByPlcActive =>, EncoderLifeValid =>, PresetBusy =>, PresetDone =>, PresetError =>, PresetStatus =>, Status =>)
   END_RUNG
   // the same network as SCL:
   "DB_EncCom_4BR1"(HW_ID_Tlg89 := "4BR1~EO_Encoder_Multiturn_V2_x_1~Standard_Telegram_89__PZD3_5",   // "FB_Enc_Tlg89_Com"
                    Enable := TRUE,
                    PresetServiceEnable := "DB_EncCtrl"."4BR1".PresetServiceEnable,
                    PresetPermit := "DB_EncCtrl"."4BR1".PresetPermit,
                    PresetStart := "DB_EncCtrl"."4BR1".PresetStart,
                    PresetValueRaw := "DB_EncCtrl"."4BR1".PresetValueRaw,
                    SimulationMode := "DB_EncCtrl"."4BR1".TestModeActive);
END_REGION

REGION Network 12: Масштабування положення енкодера #1 крана 4BR1 / Масштабування положення екнодеру підйому 1BR
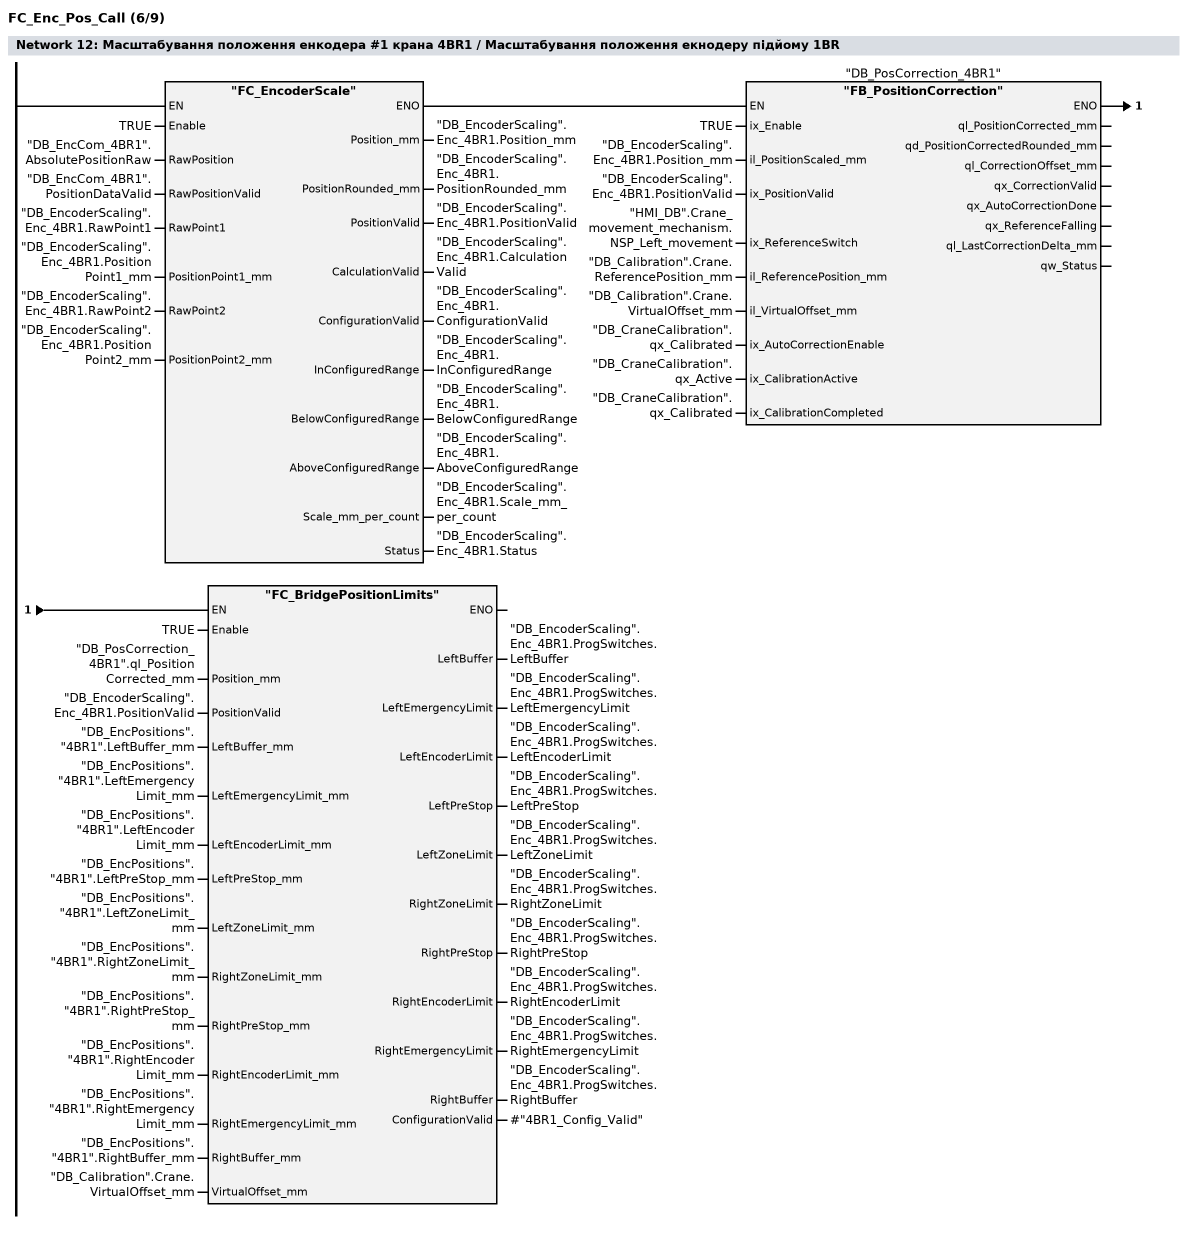
   RUNG wire#powerrail
      "FC_EncoderScale"(Enable := TRUE, RawPosition := "DB_EncCom_4BR1".AbsolutePositionRaw, RawPositionValid := "DB_EncCom_4BR1".PositionDataValid, RawPoint1 := "DB_EncoderScaling".Enc_4BR1.RawPoint1, PositionPoint1_mm := "DB_EncoderScaling".Enc_4BR1.PositionPoint1_mm, RawPoint2 := "DB_EncoderScaling".Enc_4BR1.RawPoint2, PositionPoint2_mm := "DB_EncoderScaling".Enc_4BR1.PositionPoint2_mm, Position_mm => "DB_EncoderScaling".Enc_4BR1.Position_mm, PositionRounded_mm => "DB_EncoderScaling".Enc_4BR1.PositionRounded_mm, PositionValid => "DB_EncoderScaling".Enc_4BR1.PositionValid, CalculationValid => "DB_EncoderScaling".Enc_4BR1.CalculationValid, ConfigurationValid => "DB_EncoderScaling".Enc_4BR1.ConfigurationValid, InConfiguredRange => "DB_EncoderScaling".Enc_4BR1.InConfiguredRange, BelowConfiguredRange => "DB_EncoderScaling".Enc_4BR1.BelowConfiguredRange, AboveConfiguredRange => "DB_EncoderScaling".Enc_4BR1.AboveConfiguredRange, Scale_mm_per_count => "DB_EncoderScaling".Enc_4BR1.Scale_mm_per_count, Status => "DB_EncoderScaling".Enc_4BR1.Status)
      "DB_PosCorrection_4BR1"(ix_Enable := TRUE, il_PositionScaled_mm := "DB_EncoderScaling".Enc_4BR1.Position_mm, ix_PositionValid := "DB_EncoderScaling".Enc_4BR1.PositionValid, ix_ReferenceSwitch := "HMI_DB".Crane_movement_mechanism.NSP_Left_movement, il_ReferencePosition_mm := "DB_Calibration".Crane.ReferencePosition_mm, il_VirtualOffset_mm := "DB_Calibration".Crane.VirtualOffset_mm, ix_AutoCorrectionEnable := "DB_CraneCalibration".qx_Calibrated, ix_CalibrationActive := "DB_CraneCalibration".qx_Active, ix_CalibrationCompleted := "DB_CraneCalibration".qx_Calibrated, ql_PositionCorrected_mm =>, qd_PositionCorrectedRounded_mm =>, ql_CorrectionOffset_mm =>, qx_CorrectionValid =>, qx_AutoCorrectionDone =>, qx_ReferenceFalling =>, ql_LastCorrectionDelta_mm =>, qw_Status =>)
      "FC_BridgePositionLimits"(Enable := TRUE, Position_mm := "DB_PosCorrection_4BR1".ql_PositionCorrected_mm, PositionValid := "DB_EncoderScaling".Enc_4BR1.PositionValid, LeftBuffer_mm := "DB_EncPositions"."4BR1".LeftBuffer_mm, LeftEmergencyLimit_mm := "DB_EncPositions"."4BR1".LeftEmergencyLimit_mm, LeftEncoderLimit_mm := "DB_EncPositions"."4BR1".LeftEncoderLimit_mm, LeftPreStop_mm := "DB_EncPositions"."4BR1".LeftPreStop_mm, LeftZoneLimit_mm := "DB_EncPositions"."4BR1".LeftZoneLimit_mm, RightZoneLimit_mm := "DB_EncPositions"."4BR1".RightZoneLimit_mm, RightPreStop_mm := "DB_EncPositions"."4BR1".RightPreStop_mm, RightEncoderLimit_mm := "DB_EncPositions"."4BR1".RightEncoderLimit_mm, RightEmergencyLimit_mm := "DB_EncPositions"."4BR1".RightEmergencyLimit_mm, RightBuffer_mm := "DB_EncPositions"."4BR1".RightBuffer_mm, VirtualOffset_mm := "DB_Calibration".Crane.VirtualOffset_mm, LeftBuffer => "DB_EncoderScaling".Enc_4BR1.ProgSwitches.LeftBuffer, LeftEmergencyLimit => "DB_EncoderScaling".Enc_4BR1.ProgSwitches.LeftEmergencyLimit, LeftEncoderLimit => "DB_EncoderScaling".Enc_4BR1.ProgSwitches.LeftEncoderLimit, LeftPreStop => "DB_EncoderScaling".Enc_4BR1.ProgSwitches.LeftPreStop, LeftZoneLimit => "DB_EncoderScaling".Enc_4BR1.ProgSwitches.LeftZoneLimit, RightZoneLimit => "DB_EncoderScaling".Enc_4BR1.ProgSwitches.RightZoneLimit, RightPreStop => "DB_EncoderScaling".Enc_4BR1.ProgSwitches.RightPreStop, RightEncoderLimit => "DB_EncoderScaling".Enc_4BR1.ProgSwitches.RightEncoderLimit, RightEmergencyLimit => "DB_EncoderScaling".Enc_4BR1.ProgSwitches.RightEmergencyLimit, RightBuffer => "DB_EncoderScaling".Enc_4BR1.ProgSwitches.RightBuffer, ConfigurationValid => #"4BR1_Config_Valid")
   END_RUNG
   // the same network as SCL:
   "FC_EncoderScale"(Enable := TRUE,
                     RawPosition := "DB_EncCom_4BR1".AbsolutePositionRaw,
                     RawPositionValid := "DB_EncCom_4BR1".PositionDataValid,
                     RawPoint1 := "DB_EncoderScaling".Enc_4BR1.RawPoint1,
                     PositionPoint1_mm := "DB_EncoderScaling".Enc_4BR1.PositionPoint1_mm,
                     RawPoint2 := "DB_EncoderScaling".Enc_4BR1.RawPoint2,
                     PositionPoint2_mm := "DB_EncoderScaling".Enc_4BR1.PositionPoint2_mm,
                     Position_mm => "DB_EncoderScaling".Enc_4BR1.Position_mm,
                     PositionRounded_mm => "DB_EncoderScaling".Enc_4BR1.PositionRounded_mm,
                     PositionValid => "DB_EncoderScaling".Enc_4BR1.PositionValid,
                     CalculationValid => "DB_EncoderScaling".Enc_4BR1.CalculationValid,
                     ConfigurationValid => "DB_EncoderScaling".Enc_4BR1.ConfigurationValid,
                     InConfiguredRange => "DB_EncoderScaling".Enc_4BR1.InConfiguredRange,
                     BelowConfiguredRange => "DB_EncoderScaling".Enc_4BR1.BelowConfiguredRange,
                     AboveConfiguredRange => "DB_EncoderScaling".Enc_4BR1.AboveConfiguredRange,
                     Scale_mm_per_count => "DB_EncoderScaling".Enc_4BR1.Scale_mm_per_count,
                     Status => "DB_EncoderScaling".Enc_4BR1.Status,
                     ENO => #_w1);
   "DB_PosCorrection_4BR1"(EN := #_w1,   // "FB_PositionCorrection"
                           ix_Enable := TRUE,
                           il_PositionScaled_mm := "DB_EncoderScaling".Enc_4BR1.Position_mm,
                           ix_PositionValid := "DB_EncoderScaling".Enc_4BR1.PositionValid,
                           ix_ReferenceSwitch := "HMI_DB".Crane_movement_mechanism.NSP_Left_movement,
                           il_ReferencePosition_mm := "DB_Calibration".Crane.ReferencePosition_mm,
                           il_VirtualOffset_mm := "DB_Calibration".Crane.VirtualOffset_mm,
                           ix_AutoCorrectionEnable := "DB_CraneCalibration".qx_Calibrated,
                           ix_CalibrationActive := "DB_CraneCalibration".qx_Active,
                           ix_CalibrationCompleted := "DB_CraneCalibration".qx_Calibrated,
                           ENO => #_w2);
   IF #_w2 THEN
       "FC_BridgePositionLimits"(Enable := TRUE,
                               Position_mm := "DB_PosCorrection_4BR1".ql_PositionCorrected_mm,
                               PositionValid := "DB_EncoderScaling".Enc_4BR1.PositionValid,
                               LeftBuffer_mm := "DB_EncPositions"."4BR1".LeftBuffer_mm,
                               LeftEmergencyLimit_mm := "DB_EncPositions"."4BR1".LeftEmergencyLimit_mm,
                               LeftEncoderLimit_mm := "DB_EncPositions"."4BR1".LeftEncoderLimit_mm,
                               LeftPreStop_mm := "DB_EncPositions"."4BR1".LeftPreStop_mm,
                               LeftZoneLimit_mm := "DB_EncPositions"."4BR1".LeftZoneLimit_mm,
                               RightZoneLimit_mm := "DB_EncPositions"."4BR1".RightZoneLimit_mm,
                               RightPreStop_mm := "DB_EncPositions"."4BR1".RightPreStop_mm,
                               RightEncoderLimit_mm := "DB_EncPositions"."4BR1".RightEncoderLimit_mm,
                               RightEmergencyLimit_mm := "DB_EncPositions"."4BR1".RightEmergencyLimit_mm,
                               RightBuffer_mm := "DB_EncPositions"."4BR1".RightBuffer_mm,
                               VirtualOffset_mm := "DB_Calibration".Crane.VirtualOffset_mm,
                               LeftBuffer => "DB_EncoderScaling".Enc_4BR1.ProgSwitches.LeftBuffer,
                               LeftEmergencyLimit => "DB_EncoderScaling".Enc_4BR1.ProgSwitches.LeftEmergencyLimit,
                               LeftEncoderLimit => "DB_EncoderScaling".Enc_4BR1.ProgSwitches.LeftEncoderLimit,
                               LeftPreStop => "DB_EncoderScaling".Enc_4BR1.ProgSwitches.LeftPreStop,
                               LeftZoneLimit => "DB_EncoderScaling".Enc_4BR1.ProgSwitches.LeftZoneLimit,
                               RightZoneLimit => "DB_EncoderScaling".Enc_4BR1.ProgSwitches.RightZoneLimit,
                               RightPreStop => "DB_EncoderScaling".Enc_4BR1.ProgSwitches.RightPreStop,
                               RightEncoderLimit => "DB_EncoderScaling".Enc_4BR1.ProgSwitches.RightEncoderLimit,
                               RightEmergencyLimit => "DB_EncoderScaling".Enc_4BR1.ProgSwitches.RightEmergencyLimit,
                               RightBuffer => "DB_EncoderScaling".Enc_4BR1.ProgSwitches.RightBuffer,
                               ConfigurationValid => #"4BR1_Config_Valid");
   END_IF;
END_REGION

REGION Network 15 (SCL): ====== Пересування крана - енкодер #2 (Bridge/Crane movement - encoder #2) ====== / ====== Пересування крана - енкодер #2 (Crane movement - encoder #2) ======
END_REGION

REGION Network 16: Зв'язок з енкодером #2 крана 4BR2
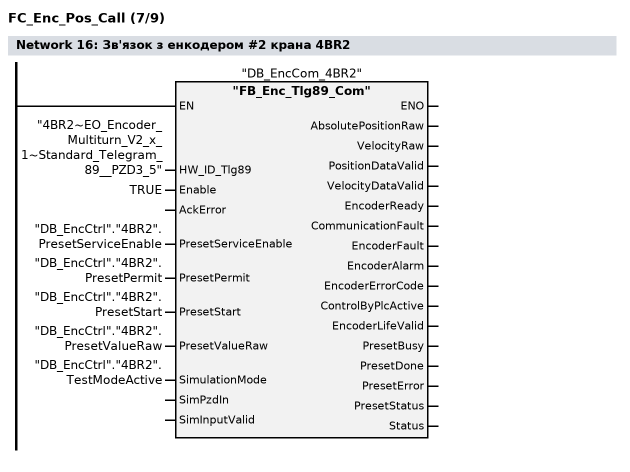
   RUNG wire#powerrail
      "DB_EncCom_4BR2"(HW_ID_Tlg89 := "4BR2~EO_Encoder_Multiturn_V2_x_1~Standard_Telegram_89__PZD3_5", Enable := TRUE, AckError :=, PresetServiceEnable := "DB_EncCtrl"."4BR2".PresetServiceEnable, PresetPermit := "DB_EncCtrl"."4BR2".PresetPermit, PresetStart := "DB_EncCtrl"."4BR2".PresetStart, PresetValueRaw := "DB_EncCtrl"."4BR2".PresetValueRaw, SimulationMode := "DB_EncCtrl"."4BR2".TestModeActive, SimPzdIn :=, SimInputValid :=, AbsolutePositionRaw =>, VelocityRaw =>, PositionDataValid =>, VelocityDataValid =>, EncoderReady =>, CommunicationFault =>, EncoderFault =>, EncoderAlarm =>, EncoderErrorCode =>, ControlByPlcActive =>, EncoderLifeValid =>, PresetBusy =>, PresetDone =>, PresetError =>, PresetStatus =>, Status =>)
   END_RUNG
   // the same network as SCL:
   "DB_EncCom_4BR2"(HW_ID_Tlg89 := "4BR2~EO_Encoder_Multiturn_V2_x_1~Standard_Telegram_89__PZD3_5",   // "FB_Enc_Tlg89_Com"
                    Enable := TRUE,
                    PresetServiceEnable := "DB_EncCtrl"."4BR2".PresetServiceEnable,
                    PresetPermit := "DB_EncCtrl"."4BR2".PresetPermit,
                    PresetStart := "DB_EncCtrl"."4BR2".PresetStart,
                    PresetValueRaw := "DB_EncCtrl"."4BR2".PresetValueRaw,
                    SimulationMode := "DB_EncCtrl"."4BR2".TestModeActive);
END_REGION

REGION Network 17: Масштабування положення енкодера #2 крана 4BR2 / Масштабування положення екнодеру підйому 1BR
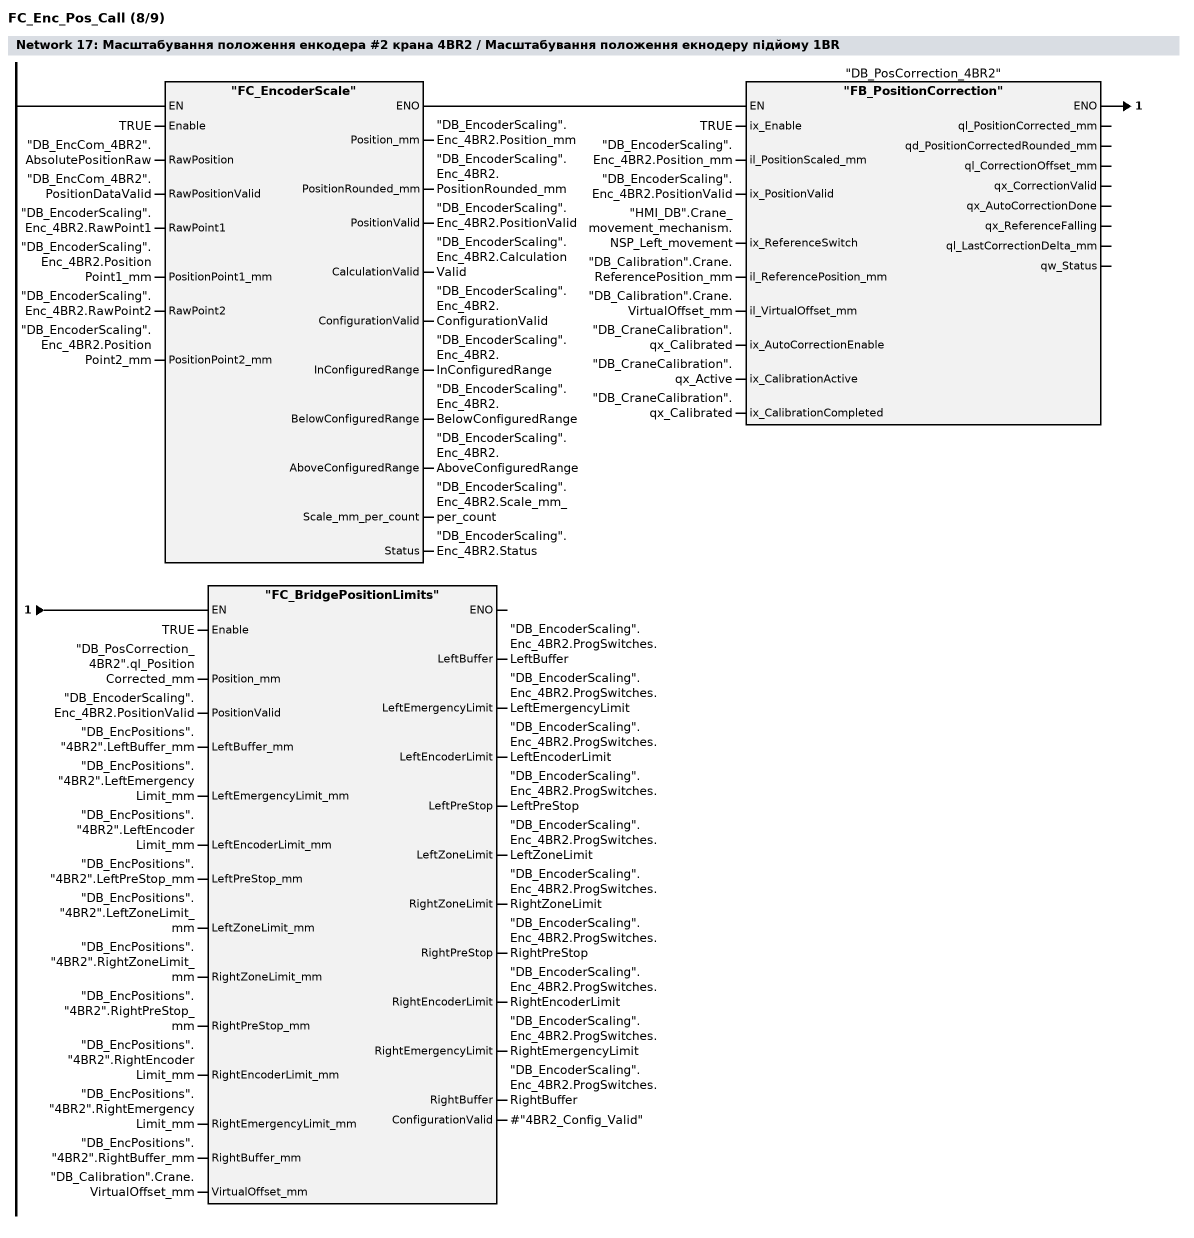
   RUNG wire#powerrail
      "FC_EncoderScale"(Enable := TRUE, RawPosition := "DB_EncCom_4BR2".AbsolutePositionRaw, RawPositionValid := "DB_EncCom_4BR2".PositionDataValid, RawPoint1 := "DB_EncoderScaling".Enc_4BR2.RawPoint1, PositionPoint1_mm := "DB_EncoderScaling".Enc_4BR2.PositionPoint1_mm, RawPoint2 := "DB_EncoderScaling".Enc_4BR2.RawPoint2, PositionPoint2_mm := "DB_EncoderScaling".Enc_4BR2.PositionPoint2_mm, Position_mm => "DB_EncoderScaling".Enc_4BR2.Position_mm, PositionRounded_mm => "DB_EncoderScaling".Enc_4BR2.PositionRounded_mm, PositionValid => "DB_EncoderScaling".Enc_4BR2.PositionValid, CalculationValid => "DB_EncoderScaling".Enc_4BR2.CalculationValid, ConfigurationValid => "DB_EncoderScaling".Enc_4BR2.ConfigurationValid, InConfiguredRange => "DB_EncoderScaling".Enc_4BR2.InConfiguredRange, BelowConfiguredRange => "DB_EncoderScaling".Enc_4BR2.BelowConfiguredRange, AboveConfiguredRange => "DB_EncoderScaling".Enc_4BR2.AboveConfiguredRange, Scale_mm_per_count => "DB_EncoderScaling".Enc_4BR2.Scale_mm_per_count, Status => "DB_EncoderScaling".Enc_4BR2.Status)
      "DB_PosCorrection_4BR2"(ix_Enable := TRUE, il_PositionScaled_mm := "DB_EncoderScaling".Enc_4BR2.Position_mm, ix_PositionValid := "DB_EncoderScaling".Enc_4BR2.PositionValid, ix_ReferenceSwitch := "HMI_DB".Crane_movement_mechanism.NSP_Left_movement, il_ReferencePosition_mm := "DB_Calibration".Crane.ReferencePosition_mm, il_VirtualOffset_mm := "DB_Calibration".Crane.VirtualOffset_mm, ix_AutoCorrectionEnable := "DB_CraneCalibration".qx_Calibrated, ix_CalibrationActive := "DB_CraneCalibration".qx_Active, ix_CalibrationCompleted := "DB_CraneCalibration".qx_Calibrated, ql_PositionCorrected_mm =>, qd_PositionCorrectedRounded_mm =>, ql_CorrectionOffset_mm =>, qx_CorrectionValid =>, qx_AutoCorrectionDone =>, qx_ReferenceFalling =>, ql_LastCorrectionDelta_mm =>, qw_Status =>)
      "FC_BridgePositionLimits"(Enable := TRUE, Position_mm := "DB_PosCorrection_4BR2".ql_PositionCorrected_mm, PositionValid := "DB_EncoderScaling".Enc_4BR2.PositionValid, LeftBuffer_mm := "DB_EncPositions"."4BR2".LeftBuffer_mm, LeftEmergencyLimit_mm := "DB_EncPositions"."4BR2".LeftEmergencyLimit_mm, LeftEncoderLimit_mm := "DB_EncPositions"."4BR2".LeftEncoderLimit_mm, LeftPreStop_mm := "DB_EncPositions"."4BR2".LeftPreStop_mm, LeftZoneLimit_mm := "DB_EncPositions"."4BR2".LeftZoneLimit_mm, RightZoneLimit_mm := "DB_EncPositions"."4BR2".RightZoneLimit_mm, RightPreStop_mm := "DB_EncPositions"."4BR2".RightPreStop_mm, RightEncoderLimit_mm := "DB_EncPositions"."4BR2".RightEncoderLimit_mm, RightEmergencyLimit_mm := "DB_EncPositions"."4BR2".RightEmergencyLimit_mm, RightBuffer_mm := "DB_EncPositions"."4BR2".RightBuffer_mm, VirtualOffset_mm := "DB_Calibration".Crane.VirtualOffset_mm, LeftBuffer => "DB_EncoderScaling".Enc_4BR2.ProgSwitches.LeftBuffer, LeftEmergencyLimit => "DB_EncoderScaling".Enc_4BR2.ProgSwitches.LeftEmergencyLimit, LeftEncoderLimit => "DB_EncoderScaling".Enc_4BR2.ProgSwitches.LeftEncoderLimit, LeftPreStop => "DB_EncoderScaling".Enc_4BR2.ProgSwitches.LeftPreStop, LeftZoneLimit => "DB_EncoderScaling".Enc_4BR2.ProgSwitches.LeftZoneLimit, RightZoneLimit => "DB_EncoderScaling".Enc_4BR2.ProgSwitches.RightZoneLimit, RightPreStop => "DB_EncoderScaling".Enc_4BR2.ProgSwitches.RightPreStop, RightEncoderLimit => "DB_EncoderScaling".Enc_4BR2.ProgSwitches.RightEncoderLimit, RightEmergencyLimit => "DB_EncoderScaling".Enc_4BR2.ProgSwitches.RightEmergencyLimit, RightBuffer => "DB_EncoderScaling".Enc_4BR2.ProgSwitches.RightBuffer, ConfigurationValid => #"4BR2_Config_Valid")
   END_RUNG
   // the same network as SCL:
   "FC_EncoderScale"(Enable := TRUE,
                     RawPosition := "DB_EncCom_4BR2".AbsolutePositionRaw,
                     RawPositionValid := "DB_EncCom_4BR2".PositionDataValid,
                     RawPoint1 := "DB_EncoderScaling".Enc_4BR2.RawPoint1,
                     PositionPoint1_mm := "DB_EncoderScaling".Enc_4BR2.PositionPoint1_mm,
                     RawPoint2 := "DB_EncoderScaling".Enc_4BR2.RawPoint2,
                     PositionPoint2_mm := "DB_EncoderScaling".Enc_4BR2.PositionPoint2_mm,
                     Position_mm => "DB_EncoderScaling".Enc_4BR2.Position_mm,
                     PositionRounded_mm => "DB_EncoderScaling".Enc_4BR2.PositionRounded_mm,
                     PositionValid => "DB_EncoderScaling".Enc_4BR2.PositionValid,
                     CalculationValid => "DB_EncoderScaling".Enc_4BR2.CalculationValid,
                     ConfigurationValid => "DB_EncoderScaling".Enc_4BR2.ConfigurationValid,
                     InConfiguredRange => "DB_EncoderScaling".Enc_4BR2.InConfiguredRange,
                     BelowConfiguredRange => "DB_EncoderScaling".Enc_4BR2.BelowConfiguredRange,
                     AboveConfiguredRange => "DB_EncoderScaling".Enc_4BR2.AboveConfiguredRange,
                     Scale_mm_per_count => "DB_EncoderScaling".Enc_4BR2.Scale_mm_per_count,
                     Status => "DB_EncoderScaling".Enc_4BR2.Status,
                     ENO => #_w1);
   "DB_PosCorrection_4BR2"(EN := #_w1,   // "FB_PositionCorrection"
                           ix_Enable := TRUE,
                           il_PositionScaled_mm := "DB_EncoderScaling".Enc_4BR2.Position_mm,
                           ix_PositionValid := "DB_EncoderScaling".Enc_4BR2.PositionValid,
                           ix_ReferenceSwitch := "HMI_DB".Crane_movement_mechanism.NSP_Left_movement,
                           il_ReferencePosition_mm := "DB_Calibration".Crane.ReferencePosition_mm,
                           il_VirtualOffset_mm := "DB_Calibration".Crane.VirtualOffset_mm,
                           ix_AutoCorrectionEnable := "DB_CraneCalibration".qx_Calibrated,
                           ix_CalibrationActive := "DB_CraneCalibration".qx_Active,
                           ix_CalibrationCompleted := "DB_CraneCalibration".qx_Calibrated,
                           ENO => #_w2);
   IF #_w2 THEN
       "FC_BridgePositionLimits"(Enable := TRUE,
                               Position_mm := "DB_PosCorrection_4BR2".ql_PositionCorrected_mm,
                               PositionValid := "DB_EncoderScaling".Enc_4BR2.PositionValid,
                               LeftBuffer_mm := "DB_EncPositions"."4BR2".LeftBuffer_mm,
                               LeftEmergencyLimit_mm := "DB_EncPositions"."4BR2".LeftEmergencyLimit_mm,
                               LeftEncoderLimit_mm := "DB_EncPositions"."4BR2".LeftEncoderLimit_mm,
                               LeftPreStop_mm := "DB_EncPositions"."4BR2".LeftPreStop_mm,
                               LeftZoneLimit_mm := "DB_EncPositions"."4BR2".LeftZoneLimit_mm,
                               RightZoneLimit_mm := "DB_EncPositions"."4BR2".RightZoneLimit_mm,
                               RightPreStop_mm := "DB_EncPositions"."4BR2".RightPreStop_mm,
                               RightEncoderLimit_mm := "DB_EncPositions"."4BR2".RightEncoderLimit_mm,
                               RightEmergencyLimit_mm := "DB_EncPositions"."4BR2".RightEmergencyLimit_mm,
                               RightBuffer_mm := "DB_EncPositions"."4BR2".RightBuffer_mm,
                               VirtualOffset_mm := "DB_Calibration".Crane.VirtualOffset_mm,
                               LeftBuffer => "DB_EncoderScaling".Enc_4BR2.ProgSwitches.LeftBuffer,
                               LeftEmergencyLimit => "DB_EncoderScaling".Enc_4BR2.ProgSwitches.LeftEmergencyLimit,
                               LeftEncoderLimit => "DB_EncoderScaling".Enc_4BR2.ProgSwitches.LeftEncoderLimit,
                               LeftPreStop => "DB_EncoderScaling".Enc_4BR2.ProgSwitches.LeftPreStop,
                               LeftZoneLimit => "DB_EncoderScaling".Enc_4BR2.ProgSwitches.LeftZoneLimit,
                               RightZoneLimit => "DB_EncoderScaling".Enc_4BR2.ProgSwitches.RightZoneLimit,
                               RightPreStop => "DB_EncoderScaling".Enc_4BR2.ProgSwitches.RightPreStop,
                               RightEncoderLimit => "DB_EncoderScaling".Enc_4BR2.ProgSwitches.RightEncoderLimit,
                               RightEmergencyLimit => "DB_EncoderScaling".Enc_4BR2.ProgSwitches.RightEmergencyLimit,
                               RightBuffer => "DB_EncoderScaling".Enc_4BR2.ProgSwitches.RightBuffer,
                               ConfigurationValid => #"4BR2_Config_Valid");
   END_IF;
END_REGION

REGION Network 18
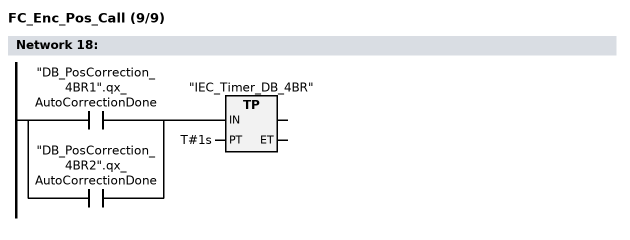
   "IEC_Timer_DB_4BR".TP(IN := "DB_PosCorrection_4BR1".qx_AutoCorrectionDone OR "DB_PosCorrection_4BR2".qx_AutoCorrectionDone,
                         PT := T#1s);
END_REGION
END_FUNCTION

FUNCTION "FC_Encoders_HMI" : Void   // FC81, SCL
{ S7_Optimized_Access := 'TRUE' }
VERSION : 0.1
BEGIN
   //Енкодер підйому
   REGION Enc_1BR
       //*********************************
       //Енкодер підйому 1BR
       //*********************************

       // ============================================================
       // Main raw values
       // ============================================================

       // Raw position from encoder G1_XIST2
       "HMI_DB".Encoders."1BR".RawPosition :=
       "DB_EncCom_1BR".AbsolutePositionRaw;

       // Raw velocity from encoder NIST_B
       "HMI_DB".Encoders."1BR".RawVelocity :=
       "DB_EncCom_1BR".VelocityRaw;


       // ============================================================
       // Main encoder status
       // ============================================================

       // Encoder is ready for crane logic
       "HMI_DB".Encoders."1BR".EncoderReady :=
       "DB_EncCom_1BR".EncoderReady;

       // Raw position is valid
       "HMI_DB".Encoders."1BR".PositionDataValid :=
       "DB_EncCom_1BR".PositionDataValid;

       // Raw velocity is valid
       "HMI_DB".Encoders."1BR".VelocityDataValid :=
       "DB_EncCom_1BR".VelocityDataValid;

       // Communication fault or cyclic data fault
       "HMI_DB".Encoders."1BR".CommunicationFault :=
       "DB_EncCom_1BR".CommunicationFault;

